// TwinCAT 3 PLC project Fraktal_Press_Demo
// Title: Fraktal_Press_Demo
// Company: fraktal-automation
// Author: fraktal-automation
// ProjectVersion: 0.1.0.10
// Description: CX2030 virtual/physical commissioning example: XTI-linked EK1200/EL1809/EL2809 HAL mapping, two-hand start, interlocked door/part slide, safety aliases, Control On/Off, AUTO/HOME/MANUAL, and model recipes.
// ProgramVersion: 3.1.4026.24
// libraries:
//   Fraktal_Core, 0.25.0.0 (fraktal-automation)
//   Fraktal_Modules, 0.11.0.3 (fraktal-automation)
//   Tc2_MC2, * (Beckhoff Automation GmbH)
//   Tc2_EtherCAT, * (Beckhoff Automation GmbH)
//   Tc2_Standard, * (Beckhoff Automation GmbH)
//   Tc2_System, * (Beckhoff Automation GmbH)
//   Tc3_Module, * (Beckhoff Automation GmbH)
// project tree:
//   00_System/Hardware/ GVL_PressIO.TcGVL, GVL_PressSafety.TcGVL
//   00_System/ GVL_PressCommissioning.TcGVL, MAIN.TcPOU, FB_PressIoDriver.TcPOU, FB_PressControlOnCircuit.TcPOU, FB_PressControlDomain.TcPOU (not stored), FB_PressOutputAuthority.TcPOU (not stored), FB_PressSimulationDriver.TcPOU (not stored)
//   01_PneumaticPress/Sequences/ FB_LD_PressDemoAuto.TcPOU, FB_PressDemoLoadPosition.TcPOU, FB_PressDemoHome.TcPOU, FB_PressDemoChangeover.TcPOU, FB_PressDemoAuto.TcPOU, FB_SFC_PressDemoAuto.TcPOU
//   / PlcTask.TcTTO (not stored)
//   01_PneumaticPress/Release/ FB_PressDemoRelease.TcPOU, FB_LD_PressDemoRelease.TcPOU, FB_PressDemoReleaseState.TcPOU
//   01_PneumaticPress/DUTs/ ST_PressDemoReleaseConditions.TcDUT, ST_PneumaticPressParCfg.TcDUT, ST_PneumaticPressStationCfg.TcDUT, ST_PneumaticPressParCmd.TcDUT (not stored), ST_PneumaticPressOutCmd.TcDUT, ST_PneumaticPressOutImm.TcDUT, E_RenditionLanguage.TcDUT
//   01_PneumaticPress/ PL_PressReasons.TcGVL, FB_PressDemoUnit.TcPOU
//   01_PneumaticPress/Recipes/ FB_PressRecipeCatalog.TcPOU
//   01_PneumaticPress/Io/ FB_PressIoCatalog.TcPOU, GVL_PressFieldbus.TcGVL
// real-time tasks:
//   TASK PlcTask: cycle T#10ms, priority 20, ADS port 350
// I/O:
//   DEVICE =000+S-A610-A1 (EtherCAT) (disabled), AmsNetId 0.0.0.0.2.1
//     =000+S-K010 (EK1200) [EK1200-5000 EtherCAT Power supply (2A E-Bus)]
//       =000+S-K010B1 (EL1809) [EL1809 16Ch. Dig. Input 24V, 3ms]
//       =000+S-K010C1 (EL2809) [EL2809 16Ch. Dig. Output 24V, 0.5A]
//       =000+S-K010D1 (EL6001) [EL6001 Interface (RS232)]
//       =000+S-K010E (EL9011) [EL9011 End Terminal]
// variable links:
//   Fraktal_Press_Demo/Fraktal_Press_Demo Instance <-> =000+S-A610-A1 (EtherCAT)/=000+S-K010 (EK1200)/=000+S-K010B1 (EL1809)
//     PlcTask Inputs/GVL_PressIO._000BS901 <-> Channel 9/_000BS901
//     PlcTask Inputs/GVL_PressIO._000BS902 <-> Channel 13/_000BS902
//     PlcTask Inputs/GVL_PressIO._000K910A <-> Channel 15/_000K910A
//     PlcTask Inputs/GVL_PressIO._000K911_Y32 <-> Channel 14/_000K911_Y32
//     PlcTask Inputs/GVL_PressIO._000MB085A_2 <-> Channel 10/_000MB085A_2
//     PlcTask Inputs/GVL_PressIO._000MB085A_4 <-> Channel 11/_000MB085A_4
//     PlcTask Inputs/GVL_PressIO._101B201A <-> Channel 3/_101B201A
//     PlcTask Inputs/GVL_PressIO._101B202A <-> Channel 5/_101B202A
//     PlcTask Inputs/GVL_PressIO._101B301A <-> Channel 1/_101B301A
//     PlcTask Inputs/GVL_PressIO._101B201B <-> Channel 4/_101B201B
//     PlcTask Inputs/GVL_PressIO._101B202B <-> Channel 6/_101B202B
//     PlcTask Inputs/GVL_PressIO._101B301B <-> Channel 2/_101B301B
//     PlcTask Inputs/GVL_PressIO._101B601 <-> Channel 12/_101B601
//     PlcTask Inputs/GVL_PressIO._101S101 <-> Channel 7/_101S101
//     PlcTask Inputs/GVL_PressIO._101S102 <-> Channel 8/_101S102
//   Fraktal_Press_Demo/Fraktal_Press_Demo Instance <-> =000+S-A610-A1 (EtherCAT)/=000+S-K010 (EK1200)/=000+S-K010C1 (EL2809)
//     PlcTask Outputs/GVL_PressIO._000K911_A1 <-> Channel 11/_000K911_A1
//     PlcTask Outputs/GVL_PressIO._000K951_A1 <-> Channel 10/_000K951_A1
//     PlcTask Outputs/GVL_PressIO._101K201A <-> Channel 3/_101K201A
//     PlcTask Outputs/GVL_PressIO._101K202A <-> Channel 5/_101K202A
//     PlcTask Outputs/GVL_PressIO._101K301A <-> Channel 1/_101K301A
//     PlcTask Outputs/GVL_PressIO._101K201B <-> Channel 4/_101K201B
//     PlcTask Outputs/GVL_PressIO._101K202B <-> Channel 6/_101K202B
//     PlcTask Outputs/GVL_PressIO._101K301B <-> Channel 2/_101K301B
//     PlcTask Outputs/GVL_PressIO._101P101 <-> Channel 7/_101P101
//     PlcTask Outputs/GVL_PressIO._101P102 <-> Channel 8/_101P102

// ---- 01_PneumaticPress/DUTs/ST_PressDemoReleaseConditions.TcDUT
// Core §7.2/§3.12 - the press's named release conditions, as PUBLISHED.
// Filled every scan from whichever rendition RELEASE_LANGUAGE selects, so a
// browsing client always reads the conditions that are actually being
// evaluated. Before this, the ST component was the published one and was
// never evaluated while LADDER_DIAGRAM was selected: every flag sat at its
// initial FALSE whatever the machine was doing - state nobody computes,
// published as if it were a claim.
TYPE ST_PressDemoReleaseConditions :
STRUCT
    ModeStartAirPressureOk : BOOL;
    RamGuardClosed    : BOOL;
    RamSlideInside    : BOOL;
    RamDevicesHealthy : BOOL;
    RamAirPressureOk  : BOOL;
    RamTwoHandHeld    : BOOL;
    RamControlPowerOn : BOOL;
END_STRUCT
END_TYPE

// ---- 01_PneumaticPress/DUTs/ST_PneumaticPressParCfg.TcDUT
// Core §3.8 ParCfg (SchemaVersion first; adding a member = schema change).
// v2 adds the §8.11 performance references: per-model ideal cycle (OEE
// Performance denominator, §8.5.1) and the WORK-time degradation baseline
// (§8.11.4(d); 0 = watch off).
//
// v3 REMOVES RequireTwoHandStart. It was recipe data in name only - every one of
// the four catalog records set it TRUE - and §3.8a's test is whether the value
// changes with the model. It does not: it answers whether this CELL's risk
// assessment demands a two-hand start, which is deployment data and now lives in
// ST_PneumaticPressStationCfg. A recipe that could switch it off would let a
// changeover quietly remove a required operator protection.
//
// TransferSettleTime deliberately STAYED. Its catalog values genuinely differ per
// model (80/100/120/150 ms): a heavier steel blank settles on the slide more
// slowly than a plastic one, so it is a fact about the part, not the mechanism.
TYPE ST_PneumaticPressParCfg :
STRUCT
    SchemaVersion       : UINT := 3;
    PressSettleTime     : TIME := T#500MS;
    TransferSettleTime  : TIME := T#100MS;
    IdealCycleMs        : UDINT := 0;    // §8.5.1 — 0 = Performance not computed
    BaselineWorkMs      : UDINT := 0;    // §8.11.4(d) — 0 = degradation watch off
END_STRUCT
END_TYPE

// ---- 01_PneumaticPress/DUTs/ST_PneumaticPressStationCfg.TcDUT
// Core §3.8a/§3.8b — what this PRESS is, as opposed to what the current product
// needs. Both members were assessed against one question: does the value change
// when the MODEL changes?
//
//   RequireTwoHandStart came OUT of ST_PneumaticPressParCfg. It was recipe data
//   in name only - all four catalog records set it TRUE - and it answers a
//   question about the CELL: does this installation's risk assessment demand a
//   two-hand start? A model recipe able to switch it off would let a changeover
//   quietly remove a required operator protection, which is not a decision a
//   product record should be able to take. (The certified two-hand evaluation
//   stays in TwinSAFE regardless, §9.8; this flag selects whether the AUTO cycle
//   WAITS for it, and can never weaken the safety function itself.)
//
//   StallGuardMs is the step guard for a step that declares no ExpectedTime
//   (§6.9). How long a pneumatic motion may take before it counts as stalled is
//   a fact about this machine's cylinders and air supply, not about the part.
//
// SchemaVersion is FIRST and mandatory (§3.8b). Version 0 means never written, so
// a first boot initializes silently; any other unrecognized version means a real
// image was rejected, and FB_ModuleBase.M_RestoreStationCfg reports it for the
// root to annunciate with this Unit's canonical path.
TYPE ST_PneumaticPressStationCfg :
STRUCT
    SchemaVersion       : UINT;    // 0 = never written; 1 = this layout
    RequireTwoHandStart : BOOL;    // cell risk-assessment policy, not recipe data
    StallGuardMs        : UDINT;   // §6.9 step guard when a step declares none
END_STRUCT
END_TYPE

// ---- 01_PneumaticPress/DUTs/ST_PneumaticPressOutCmd.TcDUT
TYPE ST_PneumaticPressOutCmd :
STRUCT
    // §3.12 — OutCmd is what a COMMAND PRODUCED, latched until the next command.
    // Both of these are genuine command results: a cycle ran, a changeover ran.
    // `Homed` used to live here and does not any more - being at the home position
    // is not something a command produced, it is something that is either true now
    // or not, so it is derived state (OutImm.Homed) recomputed every scan.
    CycleCompleted : BOOL;
    ChangeoverCompleted : BOOL;
END_STRUCT
END_TYPE

// ---- 01_PneumaticPress/DUTs/ST_PneumaticPressOutImm.TcDUT
TYPE ST_PneumaticPressOutImm :
STRUCT
    // Only facts the Unit DERIVES. A child's own state is read on the child
    // (PressRam.OutImm.Retracted, ...), never copied here under a second name (O9).
    //
    // §3.12 derived state: TRUE while the machine IS at its reference position.
    // As a latched command result it went on claiming "homed" after an operator
    // jogged an axis off home in MANUAL, because no sequence ran to clear it.
    Homed           : BOOL;
    // TRUE while a two-hand press would start a cycle: buttons armed, the control
    // domain ready, a part loaded and air present. Drives the pushbutton lamps.
    TwoHandStartReady : BOOL;
END_STRUCT
END_TYPE

// ---- 01_PneumaticPress/DUTs/E_RenditionLanguage.TcDUT
// Which language a parallel rendition of the same engineering is written in.
// The internal press bench carries the AUTO chain three times and the release
// engineering twice — the same behaviour in a second language is a
// demonstration of §5.5/§6.8 language parity, not §1.1 O9 duplication.
// FB_PressDemoUnit selects one of each; the compiler folds the branches the
// selection does not take, so the unselected renditions are inert.
//
// ONE type for both selections on purpose: a value has to mean the same
// language wherever it appears. The release engineering has no
// SEQUENTIAL_FUNCTION_CHART rendition — SFC is a sequence language and has
// nothing to say about a permissive — so that member is simply never selected
// there. The gap is deliberate; it is not an invitation to reuse the value for
// something else.
//
// The members are spelled out rather than abbreviated because 'ST' is a
// reserved word (the IL store operator). As an enumeration member it desyncs
// the parser and cascades misleading errors onto innocent lines (lint C2).
{attribute 'qualified_only'}
TYPE E_RenditionLanguage :
(
    STRUCTURED_TEXT           := 0,   // §6.8 reference form: CASE _step OF + M_Advance
    SEQUENTIAL_FUNCTION_CHART := 1,   // native XAE chart; sequences only
    LADDER_DIAGRAM            := 2    // rung-per-state integer machine over _step
) DINT;
END_TYPE

// ---- 00_System/Hardware/GVL_PressIO.TcGVL
{attribute 'qualified_only'}
// CX2030 local EtherCAT process image, reconciled with the supplied XTI export.
// TcLinkTo owns the physical link by exact terminal/channel/PDO-entry name;
// AT %I*/%Q* keeps the compiler-selected process-image offset non-positional.
VAR_GLOBAL
    // =000+S-K010B1 (EL1809) inputs
    {attribute 'TcLinkTo' := 'TIIB[=000+S-K010B1 (EL1809)]^Channel 1^_101B301A'}
    _101B301A AT %I* : BOOL;       // Ch1 feeder retracted = logical slide INSIDE
    {attribute 'TcLinkTo' := 'TIIB[=000+S-K010B1 (EL1809)]^Channel 2^_101B301B'}
    _101B301B AT %I* : BOOL;       // Ch2 feeder extended  = logical slide OUTSIDE
    {attribute 'TcLinkTo' := 'TIIB[=000+S-K010B1 (EL1809)]^Channel 3^_101B201A'}
    _101B201A AT %I* : BOOL;       // Ch3 door closed
    {attribute 'TcLinkTo' := 'TIIB[=000+S-K010B1 (EL1809)]^Channel 4^_101B201B'}
    _101B201B AT %I* : BOOL;       // Ch4 door open
    {attribute 'TcLinkTo' := 'TIIB[=000+S-K010B1 (EL1809)]^Channel 5^_101B202A'}
    _101B202A AT %I* : BOOL;       // Ch5 press down
    {attribute 'TcLinkTo' := 'TIIB[=000+S-K010B1 (EL1809)]^Channel 6^_101B202B'}
    _101B202B AT %I* : BOOL;       // Ch6 press up
    {attribute 'TcLinkTo' := 'TIIB[=000+S-K010B1 (EL1809)]^Channel 7^_101S101'}
    _101S101  AT %I* : BOOL;       // Ch7 right two-hand raw button
    {attribute 'TcLinkTo' := 'TIIB[=000+S-K010B1 (EL1809)]^Channel 8^_101S102'}
    _101S102  AT %I* : BOOL;       // Ch8 left two-hand raw button
    {attribute 'TcLinkTo' := 'TIIB[=000+S-K010B1 (EL1809)]^Channel 10^_000MB085A_2'}
    _000MB085A_2 AT %I* : BOOL;    // Ch10 compressed air below 0.3 bar
    {attribute 'TcLinkTo' := 'TIIB[=000+S-K010B1 (EL1809)]^Channel 11^_000MB085A_4'}
    _000MB085A_4 AT %I* : BOOL;    // Ch11 compressed air above 4.5 bar
    {attribute 'TcLinkTo' := 'TIIB[=000+S-K010B1 (EL1809)]^Channel 12^_101B601'}
    _101B601 AT %I* : BOOL;        // Ch12 part present
    // N54 D2 operator buttons. Free EL1809 channels were 9/13/16; 9 and 13 are
    // assigned here. The TcLinkTo names MUST match the terminal channel names in
    // XAE - confirm the physical wiring before trusting these.
    {attribute 'TcLinkTo' := 'TIIB[=000+S-K010B1 (EL1809)]^Channel 9^_000BS901'}
    _000BS901 AT %I* : BOOL;       // Ch9  IsControlOnButtonPressed  (=000+B-S901:14)
    {attribute 'TcLinkTo' := 'TIIB[=000+S-K010B1 (EL1809)]^Channel 13^_000BS902'}
    _000BS902 AT %I* : BOOL;       // Ch13 IsControlOffButtonPressed (=000+B-S902:14)
    {attribute 'TcLinkTo' := 'TIIB[=000+S-K010B1 (EL1809)]^Channel 14^_000K911_Y32'}
    _000K911_Y32 AT %I* : BOOL;    // Ch14 Control On feedback
    {attribute 'TcLinkTo' := 'TIIB[=000+S-K010B1 (EL1809)]^Channel 15^_000K910A'}
    _000K910A AT %I* : BOOL;       // Ch15 E-stop PRESSED (=000+S1-K910A:14); NORMALLY OPEN on this
                                   // demo rig: TRUE = actuated. NOT fail-safe - production needs NC.

    // =000+S-K010C1 (EL2809) outputs
    {attribute 'TcLinkTo' := 'TIIB[=000+S-K010C1 (EL2809)]^Channel 1^_101K301A'}
    _101K301A AT %Q* : BOOL;       // Ch1 feeder backward = move inside
    {attribute 'TcLinkTo' := 'TIIB[=000+S-K010C1 (EL2809)]^Channel 2^_101K301B'}
    _101K301B AT %Q* : BOOL;       // Ch2 feeder forward  = move outside
    {attribute 'TcLinkTo' := 'TIIB[=000+S-K010C1 (EL2809)]^Channel 3^_101K201A'}
    _101K201A AT %Q* : BOOL;       // Ch3 close door
    {attribute 'TcLinkTo' := 'TIIB[=000+S-K010C1 (EL2809)]^Channel 4^_101K201B'}
    _101K201B AT %Q* : BOOL;       // Ch4 open door
    {attribute 'TcLinkTo' := 'TIIB[=000+S-K010C1 (EL2809)]^Channel 5^_101K202A'}
    _101K202A AT %Q* : BOOL;       // Ch5 press downward
    {attribute 'TcLinkTo' := 'TIIB[=000+S-K010C1 (EL2809)]^Channel 6^_101K202B'}
    _101K202B AT %Q* : BOOL;       // Ch6 press upward
    {attribute 'TcLinkTo' := 'TIIB[=000+S-K010C1 (EL2809)]^Channel 7^_101P101'}
    _101P101  AT %Q* : BOOL;       // Ch7 right two-hand lamp
    {attribute 'TcLinkTo' := 'TIIB[=000+S-K010C1 (EL2809)]^Channel 8^_101P102'}
    _101P102  AT %Q* : BOOL;       // Ch8 left two-hand lamp
    {attribute 'TcLinkTo' := 'TIIB[=000+S-K010C1 (EL2809)]^Channel 10^_000K951_A1'}
    _000K951_A1 AT %Q* : BOOL;     // Ch10 SwitchControlOn functional request
    {attribute 'TcLinkTo' := 'TIIB[=000+S-K010C1 (EL2809)]^Channel 11^_000K911_A1'}
    _000K911_A1 AT %Q* : BOOL;     // Ch11 EnableControlOn functional request

    // =000+S-K010D1 (EL6001) RS232 serial interface.
    //
    // The terminal is on the bus and was previously unmapped, so it appeared in the
    // topology as a node with no channels: an operator diagnosing a dead serial link
    // had nothing to look at. Nothing in this demo speaks a serial protocol yet - the
    // process image is mapped so the card is visible, forceable and diagnosable like
    // every other node, which is what the §10.5.1 bus view is for.
    //
    // [!] NOT LINKED YET. The guessed default 3-byte PDO names (0x1A00/0x1600) were
    // wrong - XAE reports `TIIB[=000+S-K010D1 (EL6001)]^Inputs^Status` not found, so
    // this terminal is on a different PDO assignment. The variables and their §10.5.1
    // topology channels stay (the card is published and visible); only the process
    // image link is missing. To finish: open the terminal's Process Data tab, read the
    // actual PDO entry names, and restore a TcLinkTo per variable. A wrong TcLinkTo
    // fails the build loudly, which is the right failure mode - it is why these are
    // absent rather than guessed a second time.
    _000K010D1_Status AT %I* : USINT;    // serial status byte
    _000K010D1_DataIn0 AT %I* : USINT;
    _000K010D1_DataIn1 AT %I* : USINT;
    _000K010D1_DataIn2 AT %I* : USINT;
    _000K010D1_Ctrl AT %Q* : USINT;      // serial control byte
    _000K010D1_DataOut0 AT %Q* : USINT;
    _000K010D1_DataOut1 AT %Q* : USINT;
    _000K010D1_DataOut2 AT %Q* : USINT;
END_VAR

// ---- 00_System/Hardware/GVL_PressSafety.TcGVL
{attribute 'qualified_only'}
// Read-only aliases to results produced outside the standard PLC by TwinSAFE
// or a validated external safety system. They intentionally default FALSE so
// physical mode cannot energize until commissioning supplies every result.
// These variables do not themselves implement a safety function.
VAR_GLOBAL
    _EStopOk               AT %I* : BOOL;
    _GuardClosed           AT %I* : BOOL;
    _TwoHandActive         AT %I* : BOOL;
    _PneumaticPermit       AT %I* : BOOL;
    _SafetyFieldbusHealthy AT %I* : BOOL;
    _StandardIoHealthy     AT %I* : BOOL;
END_VAR

// ---- 00_System/GVL_PressCommissioning.TcGVL
{attribute 'qualified_only'}
// Deployment-owned access-provider bootstrap. Secrets deliberately have no
// source default and are excluded from OPC UA. Write a PIN here in the target's
// controlled commissioning workflow: MAIN registers it as a salted hash in the same
// scan and clears it, so no PIN is retained as text (§14). Provision users before
// locking the PLC policy.
VAR_GLOBAL PERSISTENT
    {attribute 'OPC.UA.DA' := '0'}
    OperatorPin   : STRING(32);
    {attribute 'OPC.UA.DA' := '0'}
    TechnicianPin : STRING(32);
    {attribute 'OPC.UA.DA' := '0'}
    AdminPin      : STRING(32);
END_VAR

// ---- 01_PneumaticPress/PL_PressReasons.TcGVL
{attribute 'qualified_only'}
// Core §8.8 band constants for THIS project: pneumatic press 12000-12999.
// Project codes deliberately sit outside the shipped registry, so a message
// raised with one keeps the severity and category the step chose.
VAR_GLOBAL CONSTANT
    PRESS_TWO_HAND_RELEASED : DINT := 12001;   // released mid-motion: cycle aborted, no damage
END_VAR

// ---- 01_PneumaticPress/Io/GVL_PressFieldbus.TcGVL
{attribute 'qualified_only'}
// Owner-local, bounded publication of the demo's physical CX2030 I/O tree.
// ST_IoChannel.Name is always the exact electrical-list/schematic tag.
VAR_GLOBAL
    {attribute 'OPC.UA.DA' := '1'}
    Topology : ST_FieldbusTopology;
END_VAR

// ---- 00_System/MAIN.TcPOU
// Virtual-commissioning application for one pneumatic press Unit.
// IMPORTANT: the Safe* values below simulate TwinSAFE outputs only. A deployed
// machine maps certified E-stop/two-hand/guard/safe-valve results from TwinSAFE.
PROGRAM MAIN
VAR
    RecipeCatalog : FB_PressRecipeCatalog;
    // §3.8b - WHERE this station's retained data lives is a project decision, made
    // here once: the press keeps its station, line and model data, its saved
    // parameter sets and its local users as files in DATA_FOLDER. A station with
    // no usable file system declares FB_RetainPersistMedium instead and nothing
    // else changes (users then stay in the Boot directory: a credential never goes
    // to a symbol-readable medium). On an IPC image with a write filter the folder
    // must be excluded, or every write reverts at the next boot.
    Storage : FB_FilePersistMedium;
    // §3.8b - named parameter sets on the same medium: one readable JSON-lines
    // file per saved set.
    ConfigStore : FB_MediumConfigStore;
    PartCarrier : FB_LocalPartCarrier;    // §3.16.2 BY_POSITION identity + local result ring
    AccessUsers : FB_LocalAccessProvider; // §7.7 commissioning user/PIN table
    // TF6100 TMC-Filtered publication starts at the deployed root instance.
    // The marker is inherited by PneumaticPress's published child symbols.
    {attribute 'OPC.UA.DA' := '1'}
    PneumaticPress : FB_PressDemoUnit;
    // §3.8e - the line this press stands on, and the OWNER of its data (the shift
    // calendar, §8.5.2). A line is no Unit and no module of one: it sits here,
    // beside the roots, like the control domain, and each root on the line
    // references it (SetLine) and presents its values as that root's line data.
    // A second station on this line would host a MIRROR fed through I_LineSource.
    PressLine : FB_LineDataV3;
    IoCatalog : FB_PressIoCatalog;
    IoDriver : FB_PressIoDriver;
    // Core §7.5.1 — this station's commissioning/engineering gate register.
    // Every gate below is a VAR CONSTANT of this program, so the register is
    // decided at build time and cannot be edited on a running machine. While it
    // holds anything, every root Unit carries the standing §7.5.2 annunciation.
    EngineeringMode : FB_EngineeringMode;
    ControlDomain : FB_PressControlDomain;
    OutputAuthority : FB_PressOutputAuthority;
    SimulationDriver : FB_PressSimulationDriver;
    PressHal, DoorHal, SlideHal : ST_CylinderHal;
    TwoHandHal : ST_TwoHandHal;
    PowerHal : ST_PowerGroupHal;
    PartPresentHal : ST_DigitalInputHal;
    AirPressureHal : ST_AirPressureHal;
    HealthProbe : FB_TcSystemHealthProbe;
    HealthConfig : ST_SystemHealthParCfg;
    HealthCpuLoadPct : LREAL;
    HealthMemoryAvailableMb : UDINT;
    HealthTimeSource : STRING(32);
    TaskIndex : Tc2_System.GETCURTASKINDEX;
    TaskCycleUs : UDINT;
    InitialModel : ST_ModelId;
    Plate : ST_Nameplate;
    Init : BOOL;
    // Read-only MIRRORS of the commissioning gates (see the VAR CONSTANT block).
    // They exist only so the gate state stays visible over ADS/OPC UA: the
    // compiler inlines constants, which may publish no symbol at all, and losing
    // that visibility would remove the fastest way to diagnose "no output moves".
    // They are reassigned from the constants every cycle and nothing reads them,
    // so writing one online is inert - the constant remains the only authority.
    UseSimulation : BOOL;
    ControlCircuitMappingConfirmed : BOOL;
    // §10.5.1 demand gate, written by the HMI while its fieldbus page is open.
    // FALSE parks the EtherCAT master scan (no ADS traffic for a view nobody is
    // watching); the last read states are held, never falsified.
    FieldbusViewActive : BOOL;

    // Simulation controls. E-stop is normally closed: TRUE = healthy circuit.
    SimEStopNc : BOOL := TRUE;
    SimControlOnButton : BOOL;
    SimControlOffButton : BOOL;
    SimLeftButton : BOOL;
    SimRightButton : BOOL;
    SimSafetyValveOk : BOOL := TRUE;
    SimFieldbusHealthy : BOOL := TRUE;
    SimPartPresent : BOOL := TRUE;
    SimAirPressureOk : BOOL := TRUE;
    SafeEStopOk : BOOL;
    SafeGuardClosed : BOOL;
    SafeTwoHandActive : BOOL;
    SafePneumaticPermit : BOOL;
    SafetyFieldbusHealthy : BOOL;
    StandardIoHealthy : BOOL;
    RawEStopHealthy : BOOL;
    LampsOn : BOOL;
    ControlOnEdge : R_TRIG;
    ControlOffEdge : R_TRIG;
    ControlOnAdopted : R_TRIG;   // rising edge of the relay chain's feedback
END_VAR
VAR CONSTANT
    // COMMISSIONING GATES - deliberately CONSTANT so they cannot be flipped
    // online. Defeating a gate must be a source change plus a download: a
    // reviewable, auditable act, not a live write from an HMI or ADS client.
    //
    // TRUE makes MAIN call M_ClearOutputs() every cycle, so no physical output
    // is ever energized while the simulation driver animates the plant.
    USE_SIMULATION : BOOL := FALSE;
    // FALSE makes M_WriteOutputs force _000K951_A1 and _000K911_A1 FALSE every
    // cycle. Control On then cannot energize, the hardwired N54 D2 relay chain
    // never closes, and NOTHING moves - even though the cylinder coils are
    // written unconditionally. Set TRUE only after verifying the K951/K911
    // electrical semantics on the cabinet; per N54 D2 SwitchControlOn and
    // EnableControlOn are distinct signals.
    CONTROL_CIRCUIT_MAPPING_CONFIRMED : BOOL := TRUE;
    // §G.4a - does THIS bench have a safety-rated enabling device for manual
    // motion? It does not: the Xvi is an 80 N magnetic linear motor standing on
    // the desk, outside the press. Declaring that here makes the axis's
    // StationCfg say the same thing, and the §7.5 gate below makes the machine
    // announce the departure for as long as it is true. A real cell with a
    // person inside it sets this TRUE and the §G.4a rule applies unchanged.
    JOG_ENABLE_DEVICE_REQUIRED : BOOL := FALSE;
END_VAR
VAR CONSTANT
    // §3.8b - this station's data folder (FB_FilePersistMedium, PATH_GENERIC).
    DATA_FOLDER : STRING(160) := 'C:\ProgramData\Fraktal\PressDemo\';
END_VAR

// Mirror the compile-time gates so they remain observable (see declaration).
UseSimulation := USE_SIMULATION;
ControlCircuitMappingConfirmed := CONTROL_CIRCUIT_MAPPING_CONFIRMED;

IF NOT Init THEN
    Init := TRUE;
    // Initial mechanically safe/load position: ram up, door open, slide outside.
    PressHal.RetractedFb := TRUE;
    DoorHal.RetractedFb := TRUE;
    SlideHal.RetractedFb := TRUE;
    RecipeCatalog.Setup(UnitRef := PneumaticPress);
    PneumaticPress.Setup(Name := 'PneumaticPress', PressHal := PressHal, DoorHal := DoorHal,
        SlideHal := SlideHal, TwoHandHal := TwoHandHal, PowerHal := PowerHal,
        PartPresentHal := PartPresentHal, AirPressureHal := AirPressureHal,
        Recipe := RecipeCatalog.Provider);
    PressLine.Setup(Name := 'PressLine', LineId := 'PRESS-LINE-1',
        Role := E_LineRole.OWNER, Source := 0, StaleAfterMs := 0);
    PneumaticPress.SetLine(pLine := ADR(PressLine));
    // §7.5.1 — declare this project's own gates. Passing the CONSTANT as `Active`
    // is the point: an inactive gate registers nothing, so a production build
    // publishes an empty register, annunciates nothing, and exposes no gated
    // surface at all. Passing a runtime variable here would defeat §7.5.1.
    EngineeringMode.M_Declare(Name := 'USE_SIMULATION',
        DescriptionKey := 'std.engineering.simulation', Active := USE_SIMULATION);
    EngineeringMode.M_Declare(Name := 'CONTROL_CIRCUIT_UNCONFIRMED',
        DescriptionKey := 'std.engineering.controlCircuitUnconfirmed',
        Active := NOT CONTROL_CIRCUIT_MAPPING_CONFIRMED);
    EngineeringMode.M_Declare(Name := 'JOG_ENABLE_DEVICE_NOT_REQUIRED',
        DescriptionKey := 'std.engineering.jogEnableDeviceNotRequired',
        Active := NOT JOG_ENABLE_DEVICE_REQUIRED);
    // Wiring the register also declares the framework's own OUTPUT_FORCING gate
    // from PL_FraktalEngineering, so forcing can never be armed without being
    // annunciated. It must precede IoCatalog.Setup, which reads ForcingActive to
    // decide whether any channel is published as Forceable at all.
    PneumaticPress.SetEngineeringMode(Mode := EngineeringMode);
    IoDriver.Setup(UnitRef := PneumaticPress);
    IoCatalog.Setup(UnitRef := PneumaticPress, Engineering := EngineeringMode);
    // §10.5.1 — the catalog owns the approved channel join, so it is what
    // resolves a force request; the Unit only routes an already-authorized one.
    PneumaticPress.SetIoCatalog(Catalog := IoCatalog);
    ControlDomain.Setup(UnitRef := PneumaticPress);
    SimulationDriver.Setup(PressHal := PressHal, DoorHal := DoorHal, SlideHal := SlideHal);
    InitialModel.ModelCode := 'ALUMINUM';
    PneumaticPress.SetModel(Id := InitialModel);
    Plate.ProductUri := 'urn:fraktal:demo:pneumatic-press:2026-0001';
    Plate.ManufacturerName := 'Fraktal Example Project';
    Plate.ProductDesignation := 'Pneumatic Press Training Cell';
    Plate.SerialNumber := 'PRESS-DEMO-2026-0001';
    Plate.YearOfConstruction := '2026';
    Plate.SoftwareVersion := 'Fraktal Press Demo 0.1';
    PneumaticPress.SetNameplate(Plate := Plate);
    // §8.9 standard reason metadata is generated and manifest-served by the Unit.
    // §3.16 traceability: station-local BY_POSITION serials; RFID/host substitutes later
    PartCarrier.Setup(UidPrefix := 'PRESS-2026-');
    PneumaticPress.SetPartCarrier(Carrier := PartCarrier);
    // §3.8b — the medium, then everything kept on it. Composition-root wiring, no
    // per-value glue: every capability any module in this tree registered is in
    // the station, line and model documents and in every saved set already.
    Storage.Setup(Folder := DATA_FOLDER, Where := Tc2_System.PATH_GENERIC);
    ConfigStore.Setup(Medium := Storage, KeyPrefix := 'PneumaticPress.sets');
    PneumaticPress.SetConfigStore(Store := ConfigStore);
    PneumaticPress.SetPersistMedium(Medium := Storage);
    // §3.8b — this press declares the STRICT restore policy. Its station data
    // today is the two-hand requirement and the step stall guard, and the
    // two-hand requirement is the reason: losing it would mean a machine that
    // presents itself as commissioned while no longer waiting for the start
    // control this cell's risk assessment requires. DEFAULTS_AND_ANNUNCIATE is
    // the shipped default and is right for a station whose lost values are
    // conveniences; this one's are not.
    //
    // The PartFeed axis's taught position is NOT in this set. FB_AxisCM
    // registers it (Annex G §G.4b), but PartFeed is neither bound by
    // ConfigurePartFeedAxis nor registered as a child of this Unit while no NC
    // axis exists in the System Manager — so it is outside the walk, and a
    // station set taken here does not contain it. It joins the set the day the
    // axis is linked, with no change to this line.
    PneumaticPress.SetConfigRestorePolicy(
        Policy := E_ConfigRestorePolicy.BLOCK_UNTIL_ACKNOWLEDGED);
    // §G.4a - the axis's own retained StationCfg is the authority; this states
    // the bench's fact into it. Stamps the schema version too, so the value
    // survives the axis's later Setup/restore rather than being defaulted over.
    IF NOT JOG_ENABLE_DEVICE_REQUIRED THEN
        PneumaticPress.PartFeed.SetJogRequiresEnable(Required := FALSE);
    END_IF
    // §7.7(c) - the user table (names and salted PIN hashes) on the same medium.
    AccessUsers.M_UseMedium(Medium := Storage);
    AccessUsers.M_UseKey(Key := 'PneumaticPress.users');
    PneumaticPress.Access.Setup(Provider := AccessUsers, pAlarmLog := ADR(PneumaticPress.AlarmLog));
    TaskIndex();
    TaskCycleUs := _TaskInfo[TaskIndex.index].CycleTime / 10;
    HealthConfig.MaxTaskCycleUs := TaskCycleUs + 2000;
    HealthProbe.M_UseWindowsTime(Enabled := NOT USE_SIMULATION,
        FilePath := PL_Fraktal.WINDOWS_CLOCK_SAMPLE_FILE, MaximumSampleAge := T#90S,
        MaximumSyncAgeSeconds := 7200, MaximumOffsetUs := HealthConfig.MaxTimeOffsetUs);
    // §8.12/§10.5 - the real profile measures controller/IPC health through the
    // Beckhoff Device Manager and the bus through the EtherCAT master's own state,
    // frame and CRC counters; simulation keeps the synthetic explicit inputs.
    HealthProbe.M_UseIpcDiagnostics(Enabled := NOT USE_SIMULATION);
    IF NOT USE_SIMULATION THEN
        HealthProbe.M_UseEtherCatMaster(pBus := IoDriver.M_BusHealth());
    END_IF
    HealthConfig.MaxTaskJitterUs := 2000;
    HealthConfig.RequireFieldbus := TRUE;
    HealthConfig.RequireDcSync := FALSE;
    HealthConfig.RequireTimeSync := TRUE;
END_IF

// §7.7/§14: a PIN is deployment configuration, never a source literal. Write one
// into GVL_PressCommissioning (XAE watch window) and it is registered as a salted
// hash in this scan and wiped: no PIN is retained as text, and the persistent user
// table keeps the user across restarts. Provision users before raising a threshold.
IF GVL_PressCommissioning.OperatorPin <> '' THEN
    AccessUsers.Register(User := 'operator', Pin := GVL_PressCommissioning.OperatorPin,
        Level := E_AccessLevel.OPERATOR);
    GVL_PressCommissioning.OperatorPin := '';
END_IF
IF GVL_PressCommissioning.TechnicianPin <> '' THEN
    AccessUsers.Register(User := 'tech', Pin := GVL_PressCommissioning.TechnicianPin,
        Level := E_AccessLevel.TECHNICIAN);
    GVL_PressCommissioning.TechnicianPin := '';
END_IF
IF GVL_PressCommissioning.AdminPin <> '' THEN
    AccessUsers.Register(User := 'admin', Pin := GVL_PressCommissioning.AdminPin,
        Level := E_AccessLevel.ADMIN);
    GVL_PressCommissioning.AdminPin := '';
END_IF

// Ordinary simulated local station buttons. The worksheet does not list real
// Control On/Off input buttons; physical operation therefore uses HMI requests
// until those devices are identified. Control Off wins simultaneous edges.
// Source the Control On/Off edges from the REAL buttons on a live machine, and
// from the simulated ones only under USE_SIMULATION. Previously both edges were
// ANDed with USE_SIMULATION, so on hardware neither could ever fire and the
// machine had no headless Control On path at all.
IF USE_SIMULATION THEN
    ControlOnEdge(CLK := SimControlOnButton);
    ControlOffEdge(CLK := SimControlOffButton);
ELSE
    ControlOnEdge(CLK := IoDriver.ControlOnButton);
    ControlOffEdge(CLK := IoDriver.ControlOffButton);
END_IF
IF ControlOffEdge.Q THEN
    PneumaticPress.RequestLocalControl(ControlOn := FALSE);
ELSIF ControlOnEdge.Q THEN
    PneumaticPress.RequestLocalControl(ControlOn := TRUE);
END_IF
// Adopt the relay chain's established state: it is the authority. Without this
// the PLC can sit with no power request while K911_Y32 shows control is already
// ON (observed on the press), leaving PLC and hardware permanently out of step.
// One-shot: re-issuing POWER_ON every scan would re-fault the power group on
// any momentary permit dip and spam the event log. Latch on the feedback's
// rising edge only, and re-arm the latch when control drops away.
ControlOnAdopted(CLK := PowerHal.PowerFeedback);
IF NOT USE_SIMULATION AND ControlOnAdopted.Q AND NOT ControlOffEdge.Q THEN
    PneumaticPress.RequestLocalControl(ControlOn := TRUE);
END_IF

IF USE_SIMULATION THEN
    SimulationDriver.M_ReadInputs(DoorHal := DoorHal, TwoHandHal := TwoHandHal,
        PowerHal := PowerHal, PartPresentHal := PartPresentHal,
        AirPressureHal := AirPressureHal, RawEStopHealthy := RawEStopHealthy,
        SafeEStopOk := SafeEStopOk, SafeGuardClosed := SafeGuardClosed,
        SafeTwoHandActive := SafeTwoHandActive,
        SafePneumaticPermit := SafePneumaticPermit,
        SafetyFieldbusHealthy := SafetyFieldbusHealthy,
        StandardIoHealthy := StandardIoHealthy, SimEStopNc := SimEStopNc,
        SimLeftButton := SimLeftButton, SimRightButton := SimRightButton,
        SimSafetyValveOk := SimSafetyValveOk,
        SimFieldbusHealthy := SimFieldbusHealthy,
        SimPartPresent := SimPartPresent, SimAirPressureOk := SimAirPressureOk,
        PowerRequested := PowerHal.EnableRequestOut);
ELSE
    // The project Hardware Driver is the only raw process-image consumer.
    IoDriver.M_ReadInputs(PressHal := PressHal, DoorHal := DoorHal,
        SlideHal := SlideHal, TwoHandHal := TwoHandHal, PowerHal := PowerHal,
        PartPresentHal := PartPresentHal, AirPressureHal := AirPressureHal,
        RawEStopHealthy := RawEStopHealthy, SafeEStopOk := SafeEStopOk,
        SafeGuardClosed := SafeGuardClosed, SafeTwoHandActive := SafeTwoHandActive,
        SafePneumaticPermit := SafePneumaticPermit,
        SafetyFieldbusHealthy := SafetyFieldbusHealthy,
        StandardIoHealthy := StandardIoHealthy);
END_IF
TwoHandHal.SafeActive := SafeTwoHandActive;
TwoHandHal.FieldbusHealthy := SafetyFieldbusHealthy;
PowerHal.SafetyPermit := SafePneumaticPermit;
PowerHal.FieldbusHealthy := StandardIoHealthy;

ControlDomain.M_Update(SafeEStopOk := SafeEStopOk,
    SafeGuardClosed := SafeGuardClosed, SafeTwoHandActive := SafeTwoHandActive,
    SafePneumaticPermit := SafePneumaticPermit,
    SafetyFieldbusHealthy := SafetyFieldbusHealthy,
    StandardIoHealthy := StandardIoHealthy, RawEStopHealthy := RawEStopHealthy,
    PowerFeedback := PowerHal.PowerFeedback,
    PowerRequested := PowerHal.EnableRequestOut,
    TwoHandFieldbusHealthy := TwoHandHal.FieldbusHealthy);
PneumaticPress.ControlDomain := ControlDomain.Status;

// §2.7/§8.12: in the real profile the probe measures the target itself - Windows
// Time through the local observer, controller/IPC metrics through the Device
// Manager, the bus through the EtherCAT master - and those groups ignore the
// explicit inputs below, which remain the simulation profile's synthetic values.
IF USE_SIMULATION THEN
    HealthCpuLoadPct := 25.0;
    HealthMemoryAvailableMb := UDINT#1024;
    HealthTimeSource := 'SIMULATED';
ELSE
    HealthCpuLoadPct := 0.0;
    HealthMemoryAvailableMb := UDINT#0;
    HealthTimeSource := 'WINDOWS/W32TIME';
END_IF
TaskIndex();
TaskCycleUs := _TaskInfo[TaskIndex.index].CycleTime / 10;
HealthProbe.Cyclic(ExpectedCycleUs := TaskCycleUs,
    ExternalTaskOverrun := _TaskInfo[TaskIndex.index].CycleTimeExceeded,
    ControllerAvailable := USE_SIMULATION,
    CpuLoadPct := HealthCpuLoadPct,
    MemoryAvailableMb := HealthMemoryAvailableMb,
    IpcAvailable := FALSE, IpcTemperatureC := 0.0,
    FanHealthy := TRUE, StorageHealthPct := 100.0,
    FieldbusAvailable := TRUE, FieldbusMasterHealthy := StandardIoHealthy,
    LostFrameCount := 0, SlaveErrorCount := 0,
    DcAvailable := USE_SIMULATION, DcSynchronized := USE_SIMULATION,
    TimeAvailable := USE_SIMULATION, TimeSynchronized := USE_SIMULATION,
    TimeSource := HealthTimeSource,
    TimeOffsetUs := 0, LastSyncAt := F_Now());
IF HealthProbe.Health.TaskAvailable THEN
    PneumaticPress.SetSystemHealth(Input := HealthProbe.Health, ParCfg := HealthConfig);
ELSE
    ; // first monotonic sample has no prior scan from which to derive a period
END_IF

// First execute ordinary control, then apply a standard-PLC withdrawal layer.
// This is defense in depth only: the real safety system owns pneumatic removal.
PneumaticPress();
OutputAuthority.M_Apply(PressHal := PressHal, DoorHal := DoorHal,
    SlideHal := SlideHal, PowerFeedback := PowerHal.PowerFeedback,
    SafePneumaticPermit := SafePneumaticPermit,
    StandardIoHealthy := StandardIoHealthy,
    HazardousRamPermit := SafeGuardClosed AND SafeTwoHandActive);
IF USE_SIMULATION THEN
    // Never leave physical outputs energized while virtual commissioning.
    IoDriver.M_ClearOutputs();
    SimulationDriver.M_RefreshPlant();
ELSE
    LampsOn := PneumaticPress.OutImm.TwoHandStartReady;
    IoDriver.M_WriteOutputs(PressHal := PressHal, DoorHal := DoorHal,
        SlideHal := SlideHal, PowerHal := PowerHal, LampsOn := LampsOn,
        ControlCircuitMappingConfirmed := CONTROL_CIRCUIT_MAPPING_CONFIRMED,
        ForcePermitted := PneumaticPress.M_ForcePermitted());
END_IF
// Node state comes from the real EtherCAT master. §10.5.1 is a diagnostic
// surface, so the master is scanned only while a client is watching the bus
// view: the HMI sets FieldbusViewActive when its fieldbus page is open (the same
// on-demand gating the read tiers already apply to the topology data itself).
IoDriver.M_RefreshFieldbus(BusViewActive := FieldbusViewActive);

END_PROGRAM

// ---- 01_PneumaticPress/Recipes/FB_PressRecipeCatalog.TcPOU
// Owner-local recipe engineering data: model identities and their typed Unit records.
// Generic validation/storage remains in FB_LocalRecipeProvider; process behavior
// remains in the project-owned FB_PressDemoUnit. MAIN only composes the two.
FUNCTION_BLOCK FB_PressRecipeCatalog
VAR_OUTPUT
    {attribute 'OPC.UA.DA' := '0'}
    Provider : FB_LocalRecipeProvider;
END_VAR
VAR PERSISTENT
    // §3.8b - the records are edited through the Unit's model data (any model;
    // the provider's Save writes here) and must outlive a restart, so they are
    // retained and seeded only once.
    _default : ST_PneumaticPressParCfg;
    _aluminum : ST_PneumaticPressParCfg;
    _plastic : ST_PneumaticPressParCfg;
    _steel : ST_PneumaticPressParCfg;
    _seeded : UINT;               // RECIPE_SEED once the defaults below were written
END_VAR
VAR
    _model : ST_ModelId;
    _configured : BOOL;
END_VAR
VAR CONSTANT
    // Bump to re-seed every record with the design values below (a download that
    // changes them, or a record layout change).
    RECIPE_SEED : UINT := 1;
END_VAR

// Static catalog: no cyclic work.

METHOD Setup : BOOL
VAR_INPUT
    UnitRef : REFERENCE TO FB_PressDemoUnit;
END_VAR
VAR
    Ok : BOOL;
END_VAR
IF _configured THEN
    Setup := TRUE;
    RETURN;
END_IF

// §8.11 per-model performance references: IdealCycleMs feeds OEE Performance
// (§8.5.1); BaselineWorkMs arms the WORK-time degradation watch (§8.11.4(d)).
// Values = design cycle for this training cell (motions + settle + dwell).
// Seeded once: afterwards the retained records hold what was edited.
IF _seeded <> RECIPE_SEED THEN
    _default.PressSettleTime := T#500MS;
    _default.TransferSettleTime := T#100MS;
    _default.IdealCycleMs := 6000;
    _default.BaselineWorkMs := 6000;
    _aluminum.PressSettleTime := T#300MS;
    _aluminum.TransferSettleTime := T#80MS;
    _aluminum.IdealCycleMs := 5700;
    _aluminum.BaselineWorkMs := 5700;
    _plastic.PressSettleTime := T#650MS;
    _plastic.TransferSettleTime := T#120MS;
    _plastic.IdealCycleMs := 6200;
    _plastic.BaselineWorkMs := 6200;
    _steel.PressSettleTime := T#1200MS;
    _steel.TransferSettleTime := T#150MS;
    _steel.IdealCycleMs := 6800;
    _steel.BaselineWorkMs := 6800;
    _seeded := RECIPE_SEED;
END_IF

Ok := Provider.Register(ModelCode := '', RecipeKey := 'PneumaticPressUnit',
    pData := ADR(_default), Size := SIZEOF(_default));
Ok := Provider.Register(ModelCode := 'ALUMINUM', RecipeKey := 'PneumaticPressUnit',
    pData := ADR(_aluminum), Size := SIZEOF(_aluminum)) AND Ok;
Ok := Provider.Register(ModelCode := 'PLASTIC', RecipeKey := 'PneumaticPressUnit',
    pData := ADR(_plastic), Size := SIZEOF(_plastic)) AND Ok;
Ok := Provider.Register(ModelCode := 'STEEL', RecipeKey := 'PneumaticPressUnit',
    pData := ADR(_steel), Size := SIZEOF(_steel)) AND Ok;

_model.ModelCode := 'ALUMINUM';
Ok := UnitRef.RegisterAvailableModel(Id := _model) AND Ok;
_model.ModelCode := 'PLASTIC';
Ok := UnitRef.RegisterAvailableModel(Id := _model) AND Ok;
_model.ModelCode := 'STEEL';
Ok := UnitRef.RegisterAvailableModel(Id := _model) AND Ok;

_configured := Ok;
Setup := Ok;
END_METHOD

END_FUNCTION_BLOCK

// ---- 01_PneumaticPress/FB_PressDemoUnit.TcPOU
// Project-owned Unit: pneumatic press + access door + transfer slide + two-hand request.
// Cylinder interlocks prevent the two documented collisions in AUTO and MANUAL.
// Certified E-stop, two-hand evaluation and safe valve outputs remain external.
FUNCTION_BLOCK FB_PressDemoUnit EXTENDS FB_UnitBase
VAR_INPUT
    ParCfg : ST_PneumaticPressParCfg;
    ParCmd : ST_PneumaticPressParCmd;
END_VAR
VAR_OUTPUT
    PressRam      : FB_CylinderCM;
    Door          : FB_CylinderCM;
    PartSlide     : FB_CylinderCM;
    TwoHand       : FB_TwoHandStartCM;
    PneumaticPower: FB_PowerGroupCM;
    PartPresentSensor : FB_DigitalInputCM;
    AirPressureMonitor : FB_AirPressureMonitorCM;
    // Jenny Science XENAX Xvi servo (Annex G, PLCopen Motion). NOT CABINET
    // HARDWARE - read the note on PartFeedAxis before looking for it there.
    PartFeed      : FB_AxisCM;
    // Project-owned, browseable condition state of the rendition that RUNS.
    ReleaseConditions : ST_PressDemoReleaseConditions;
    OutCmd        : ST_PneumaticPressOutCmd;
    OutImm        : ST_PneumaticPressOutImm;
END_VAR
VAR
    {attribute 'OPC.UA.DA' := '0'}
    _recipe : I_RecipeProvider;
    // The NC axis this Unit feeds parts with. Until an axis is actually linked
    // in the System Manager, _partFeedConfigured stays FALSE and the module is
    // never called: MC_Power against an unlinked AXIS_REF would otherwise run
    // every scan on a bench whose eight tests are green. Absent hardware is
    // absent, not silently pretended.
    //
    // WHAT THIS AXIS IS, AND IS NOT (2026-08-25). The delivered CX2030 cabinet
    // has NO SERVO. Its approved I/O list is five Beckhoff terminals
    // (=000+S-K010: EK1200 / EL1809 / EL2809 / EL6001 / EL9011 -- see
    // Specification/Reports/CX2030_PRESS_IO_MAPPING.md), and the part feeder in
    // that cabinet is PNEUMATIC: PartSlide above, driven by the digital outputs
    // _101K301A/_101K301B. Do not go looking for this axis on the cabinet bus.
    //
    // The drive behind it is a Jenny Science XENAX Xvi (vendor #x557, product
    // #x7508) on a SECOND EtherCAT device, =000+S-A620 (EtherCAT), kept in its
    // own XTI beside the cabinet's. It is outside the press entirely and stands
    // in for a feed axis so a real process can be simulated against real motion
    // hardware. Anything it teaches (S3.8c) or persists (S3.8b) is BENCH data,
    // not commissioning data for the press -- which is why =000+S-A610-A1
    // (EtherCAT).xti, the faithful record of the delivered cabinet, does not
    // mention it and must not be made to.
    {attribute 'OPC.UA.DA' := '0'}
    PartFeedAxis : AXIS_REF;
    _partFeedConfigured : BOOL;
    _partFeedArmed : BOOL;             // last arming attempt's result (S5.6: no discarded return)
    // §10.5.1 - the project I/O catalog owns the approved channel identity join
    // (§10.2.1), so it, not this Unit, resolves a force request to a physical
    // channel. Absent = no force routing, which is the fail-closed default.
    {attribute 'OPC.UA.DA' := '0'}
    _ioCatalog : REFERENCE TO FB_PressIoCatalog;
    _parCfgStaged : ST_PneumaticPressParCfg;
    // §3.8a - the ParCfg last applied (commit or accepted edit); a difference is an
    // edit of the active model's recipe to take effect and to write back.
    {attribute 'OPC.UA.DA' := '0'}
    _parCfgApplied : ST_PneumaticPressParCfg;
    _recipePrepared : BOOL;
    _startLatched : BOOL;
    _powerRequestPending : BOOL;
    _powerTargetOn : BOOL;
    {attribute 'OPC.UA.DA' := '0'}
    _homeSequence : FB_PressDemoHome;       // §6.8 ST chain on FB_SequenceBase owns HOME steps
    {attribute 'OPC.UA.DA' := '0'}
    _changeoverSequence : FB_PressDemoChangeover;
    // §6.8 / O2 — the SAME AUTO chain in all three permitted languages. This is a
    // demo bench: carrying three renditions is the point (O2 says sequences and
    // interlocks may be ST, SFC or Ladder), not something a real project would do.
    // AUTO_SEQUENCE_LANGUAGE below picks which one the Unit binds and runs; the
    // other two are inert. They are excluded from OPC UA for the same reason the
    // bound one is: a chain is not a module and publishes no Status.
    {attribute 'OPC.UA.DA' := '0'}
    _autoSequence : FB_PressDemoAuto;
    {attribute 'OPC.UA.DA' := '0'}
    _sfcAutoSequence : FB_SFC_PressDemoAuto;
    {attribute 'OPC.UA.DA' := '0'}
    _ldAutoSequence : FB_LD_PressDemoAuto;
    // §7.2 / O2 — the SAME release engineering in a second language. Only the
    // rendition RELEASE_LANGUAGE selects is set up, evaluated, and allowed to
    // write the directional permits and the release report; the other is inert.
    // Neither rendition is published itself: the selected one fills
    // ReleaseConditions (a VAR_OUTPUT above) every scan, so the browseable
    // record is always the one being evaluated. Publishing the ST instance
    // directly left it frozen at FALSE whenever LD was selected (§3.12).
    {attribute 'OPC.UA.DA' := '0'}
    _stReleaseConditions : FB_PressDemoRelease;
    {attribute 'OPC.UA.DA' := '0'}
    _ldReleaseConditions : FB_LD_PressDemoRelease;
END_VAR
VAR PERSISTENT
    // §3.8b - this station's deployment data. PERSISTENT is the BACKING, not the
    // architecture: the values are reached as (Scope, WriteKey) capabilities like
    // every other editable value, never as an aggregate copied in and out.
    _station : ST_PneumaticPressStationCfg;
END_VAR
VAR CONSTANT
    // §3.8b - layout version of the retained image above. Bump it when a member
    // is added, and the old image is rejected and annunciated instead of read by
    // field position.
    PRESS_STATIONCFG_SCHEMA : UINT := 1;
    // §3.8 - the longest settle times a recipe may hold. ONE source for the check
    // a changeover applies (PrepareRecipe) and the range an edit is offered
    // (the PAR_CFG registration), so an edit can never store what a changeover
    // would refuse.
    RECIPE_MAX_PRESS_SETTLE_MS    : UDINT := 30000;
    RECIPE_MAX_TRANSFER_SETTLE_MS : UDINT := 5000;
    // The provider key of this Unit's recipe record: loaded at a changeover and
    // edited per model through the same key (§3.8a).
    PRESS_RECIPE_KEY : STRING(80) := 'PneumaticPressUnit';
    // Which rendition of the AUTO chain runs. VAR CONSTANT on purpose, like the
    // §6.0 commissioning gates in MAIN: switching language is a source edit plus a
    // download, never an online write. The compiler folds the unselected branches.
    //   STRUCTURED_TEXT           -> FB_PressDemoAuto
    //   SEQUENTIAL_FUNCTION_CHART -> FB_SFC_PressDemoAuto
    //   LADDER_DIAGRAM            -> FB_LD_PressDemoAuto
    AUTO_SEQUENCE_LANGUAGE : E_RenditionLanguage := E_RenditionLanguage.LADDER_DIAGRAM;
    // Which rendition of the release/interlock logic is evaluated, on the same
    // terms and from the same type, so a value means the same language in both
    // selections. There is no SEQUENTIAL_FUNCTION_CHART rendition here: SFC is a
    // sequence language and has nothing to say about a permissive, so that
    // member is simply never selected rather than being given a second meaning.
    //   STRUCTURED_TEXT -> FB_PressDemoRelease
    //   LADDER_DIAGRAM  -> FB_LD_PressDemoRelease
    RELEASE_LANGUAGE : E_RenditionLanguage := E_RenditionLanguage.LADDER_DIAGRAM;
END_VAR

Cyclic();

// §7.8 mode-entry release owned by this Unit. The base Start method consumes the
// same report the HMI displays, so this condition cannot become explanation-only.
METHOD PROTECTED _M_AppendInterlocks
VAR_IN_OUT
    Report : ST_ReleaseReport;
END_VAR
IF ModeActive <> E_Mode.CHANGEOVER THEN
IF RELEASE_LANGUAGE = E_RenditionLanguage.LADDER_DIAGRAM THEN
    _ldReleaseConditions.M_AppendStart(Report := Report);
ELSE
    _stReleaseConditions.M_AppendStart(Report := Report);
END_IF
END_IF
END_METHOD

METHOD PROTECTED _M_AppendManualInterlocks
VAR_INPUT
    TargetPath : STRING(255);
    Value : DINT;
END_VAR
VAR_IN_OUT
    Report : ST_ReleaseReport;
END_VAR
IF RELEASE_LANGUAGE = E_RenditionLanguage.LADDER_DIAGRAM THEN
    _ldReleaseConditions.M_AppendManual(TargetPath := TargetPath, Value := Value,
        PressRam := PressRam, Door := Door, PartSlide := PartSlide, Report := Report);
ELSE
    _stReleaseConditions.M_AppendManual(TargetPath := TargetPath, Value := Value,
        PressRam := PressRam, Door := Door, PartSlide := PartSlide, Report := Report);
END_IF
END_METHOD

// Clear state that must not survive init, mode entry, or either abort path. The
// base already restarts the chains and clears their decision (§6.8); this is the
// Unit's OWN state. OnCommandStart deliberately does not call this: a physical
// start pulse may have been latched one scan before the Execute edge is consumed.
METHOD PROTECTED _M_ClearModeTransitionState
_startLatched := FALSE;
END_METHOD

// Thin mode router. Each supported sequence is a named method in the Unit tree.
METHOD PROTECTED _M_Dispatch
CASE ModeActive OF
    E_Mode.AUTO:
        _M_SequenceAuto();
    E_Mode.HOME:
        _M_SequenceHome();
    E_Mode.CHANGEOVER:
        _M_SequenceChangeover();
    E_Mode.MANUAL:
        _M_Fault(E_Reason.UNSUPPORTED_COMMAND, 'project.error.pressManualHasNoSequence');
ELSE
    _M_Fault(E_Reason.UNSUPPORTED_COMMAND, 'project.error.pressModeHasNoSequence');
END_CASE
END_METHOD

// §10.2.1 — inject this station's I/O catalog so §10.5.1 force requests can be
// resolved against the approved engineering-data join instead of against a
// second copy of the channel map. Wired once by the composition root.
METHOD SetIoCatalog
VAR_INPUT
    Catalog : REFERENCE TO FB_PressIoCatalog;
END_VAR
_ioCatalog REF= Catalog;
END_METHOD

// §10.5.1 — resolve an accepted force request onto a physical output channel.
// FB_UnitBase.ForceChannel has already proved the §7.7 MANUAL access level, the
// §7.5 OUTPUT_FORCING build gate, and that this Unit is idle in MANUAL; the
// catalog then proves what only it knows — that the path names a channel of THIS
// root, that it is an OUTPUT, and that the project marked it forceable.
METHOD PROTECTED _M_RouteForceChannel : BOOL
VAR_INPUT
    ChannelPath : STRING(255);
    Force       : BOOL;
    BoolText    : STRING(255);
    AnalogText  : STRING(160);
END_VAR
_M_RouteForceChannel := FALSE;
IF NOT __ISVALIDREF(_ioCatalog) THEN
    RETURN;
END_IF
// The transported value is text (the mailbox carries no variant), so a malformed
// payload must decode to a defined value rather than to whatever the converter
// leaves behind: anything that is not exactly 'true' is FALSE (§5.6).
_M_RouteForceChannel := _ioCatalog.M_RouteForce(ChannelPath := ChannelPath,
    OwnerRootPath := _name, Force := Force,
    BoolValue := (BoolText = 'true'),
    AnalogValue := STRING_TO_REAL(AnalogText));
END_METHOD

// Wiring-only AUTO adapter. Every production command, wait, timer, decision,
// traceability action, and transition lives in the §6.8 chain.
METHOD PROTECTED _M_SequenceAuto
// An ST chain's body is a method (M_Run); an SFC or LD chain's body IS the chart,
// so the instance itself is the call. That asymmetry is the language difference,
// not an inconsistency to normalise away.
IF AUTO_SEQUENCE_LANGUAGE = E_RenditionLanguage.LADDER_DIAGRAM THEN
    _ldAutoSequence();
ELSIF AUTO_SEQUENCE_LANGUAGE = E_RenditionLanguage.SEQUENTIAL_FUNCTION_CHART THEN
    _sfcAutoSequence();
ELSE
    _autoSequence.M_Run();
END_IF
END_METHOD

// Wiring-only CHANGEOVER adapter. The §6.8 chain owns model validation, safe
// positioning, the operator decision, and completion logic.
METHOD PROTECTED _M_SequenceChangeover
_changeoverSequence.M_Run();
END_METHOD

// Wiring-only HOME adapter. OnCommandStart owns the reset edge; the sequence POU
// owns every process step and terminal action.
METHOD PROTECTED _M_SequenceHome
_homeSequence.M_Run();
END_METHOD

METHOD PROTECTED _M_Supports : BOOL
VAR_INPUT
    Mode : E_Mode;
END_VAR
_M_Supports := (Mode = E_Mode.AUTO) OR (Mode = E_Mode.MANUAL)
    OR (Mode = E_Mode.HOME) OR (Mode = E_Mode.CHANGEOVER);
END_METHOD

// §3.4.2 — the press paces every motion boundary through _M_StepGate, so
// SINGLE_STEP and HOLD_TO_RUN are supported (NON-SAFETY pacing; interlocks
// and the certified safety layer are unaffected).
METHOD PROTECTED _M_SupportsRunStyle : BOOL
VAR_INPUT
    Style : E_RunStyle;
END_VAR
_M_SupportsRunStyle := (Style = E_RunStyle.CONTINUOUS)
    OR (Style = E_RunStyle.SINGLE_STEP) OR (Style = E_RunStyle.HOLD_TO_RUN);
END_METHOD

// One safe-stop wiring point shared by normal and error-state abort transitions.
METHOD PROTECTED _M_WithdrawSequenceOutputs
PressRam.WithdrawOutputs();
Door.WithdrawOutputs();
PartSlide.WithdrawOutputs();
PressRam.Execute := FALSE;
Door.Execute := FALSE;
PartSlide.Execute := FALSE;
END_METHOD

METHOD AbortRecipe
SUPER^.AbortRecipe();
_recipePrepared := FALSE;
END_METHOD

METHOD CommitRecipe
SUPER^.CommitRecipe();
IF _recipePrepared THEN
    ParCfg := _parCfgStaged;
    // §8.11 performance references follow the model: OEE Performance denominator
    // and the WORK-time degradation baseline are per-recipe engineering data.
    Oee.IdealCycleMs := ParCfg.IdealCycleMs;
    Profiler.M_SetBaselineWork(WorkMs := ParCfg.BaselineWorkMs);
    _parCfgApplied := ParCfg;
END_IF
_recipePrepared := FALSE;
END_METHOD

// §3.10.2 — base walk (Unit facets + all child modules), then the project-owned
// fieldbus topology identity, from the I/O catalog that owns it (SetIoCatalog):
// its static members are OPC.UA.DA=0 and reach the HMI only through this manifest.
METHOD M_AppendConfig : BOOL
VAR_INPUT
    Pager : REFERENCE TO FB_ConfigPager;
END_VAR
M_AppendConfig := SUPER^.M_AppendConfig(Pager := Pager);
IF __ISVALIDREF(_ioCatalog) THEN
    _ioCatalog.M_AppendTopologyConfig(Pager := Pager);
END_IF
END_METHOD

METHOD PROTECTED OnAbort : DINT
OnAbort := SUPER^.OnAbort();
_M_PartAborted();                    // §3.16.3: the part leaves without a valid result
_M_WithdrawSequenceOutputs();
_M_ClearModeTransitionState();
_powerTargetOn := FALSE;
_powerRequestPending := TRUE;
END_METHOD

// Error-state Abort is a deliberate recovery action but does not clear ERROR.
METHOD PROTECTED OnAbortInError : DINT
OnAbortInError := SUPER^.OnAbortInError();
_M_WithdrawSequenceOutputs();
_M_ClearModeTransitionState();
_powerTargetOn := FALSE;
_powerRequestPending := TRUE;
END_METHOD

// The press's restart policy (§6.9(d)): every accepted Start gets a fresh mode
// chain, including a repeated HOME/CHANGEOVER run that does not pass through
// another mode change. Resuming where an error stopped is the other legitimate
// choice; this station does not make it.
METHOD PROTECTED OnCommandStart : DINT
OnCommandStart := SUPER^.OnCommandStart();
_M_RestartSequences();
END_METHOD

METHOD PROTECTED OnCyclic : DINT
VAR
    started : BOOL;
END_VAR
OnCyclic := SUPER^.OnCyclic();
// §3.8b/§3.12 — the step guard is DERIVED from the station value every scan, not
// latched at Setup. An operator who edits press.stallGuardMs gets the new guard
// on the next step, and the published StallTime can never disagree with the
// configuration it came from.
StallTime := UDINT_TO_TIME(_station.StallGuardMs);
// §3.8a - an accepted edit of the ACTIVE model's recipe lands in ParCfg (the base
// has already saved it to the model's record). The performance references follow
// it, as they do at a changeover.
IF MEMCMP(ADR(ParCfg), ADR(_parCfgApplied), SIZEOF(ParCfg)) <> 0 THEN
    Oee.IdealCycleMs := ParCfg.IdealCycleMs;
    Profiler.M_SetBaselineWork(WorkMs := ParCfg.BaselineWorkMs);
    _parCfgApplied := ParCfg;
END_IF
// §7.2.1/§6.1 - a cylinder cannot move without air, so air is each cylinder's own
// process condition. Lost mid-stroke, the cylinder HOLDS - outputs off, resumes by
// itself when pressure returns - and the Unit rolls the hold up by name. Nothing
// to reset: the process restores this condition, it is not a defect.
PressRam.SetAreaSafe(Ok := AirPressureMonitor.OutImm.PressureOk,
    DescriptionKey := 'project.interlock.pressRequiresAirPressure');
Door.SetAreaSafe(Ok := AirPressureMonitor.OutImm.PressureOk,
    DescriptionKey := 'project.interlock.pressRequiresAirPressure');
PartSlide.SetAreaSafe(Ok := AirPressureMonitor.OutImm.PressureOk,
    DescriptionKey := 'project.interlock.pressRequiresAirPressure');
// Project release engineering is a separate visible component. It owns the
// functional collision permits and mode-entry conditions consumed below.
IF RELEASE_LANGUAGE = E_RenditionLanguage.LADDER_DIAGRAM THEN
    _ldReleaseConditions.M_Evaluate(PressRam := PressRam, Door := Door, PartSlide := PartSlide,
        TwoHand := TwoHand, PneumaticPower := PneumaticPower,
        AirPressure := AirPressureMonitor);
    _ldReleaseConditions.M_PublishTo(Conditions := ReleaseConditions);
ELSE
    _stReleaseConditions.M_Evaluate(PressRam := PressRam, Door := Door, PartSlide := PartSlide,
        TwoHand := TwoHand, PneumaticPower := PneumaticPower,
        AirPressure := AirPressureMonitor);
    _stReleaseConditions.M_PublishTo(Conditions := ReleaseConditions);
END_IF

// S1.1 O1 - the axis ARMS ITSELF on the first scan a real NC axis is behind
// it, rather than through a call a composition root has to remember. Forgetting
// such a call produces a silently dead module, which is exactly the class of
// defect the objective says to drive from a path the application already takes.
// ConfigurePartFeedAxis is idempotent and fails closed, so calling it until it
// succeeds costs one comparison per scan on a bench with no drive.
IF NOT _partFeedConfigured THEN
    // THIS^ is required: an unqualified same-FB call resolves only when its
    // return value is discarded, and this one is not (C0009/C0035 otherwise).
    _partFeedArmed := THIS^.ConfigurePartFeedAxis(AxisRef := PartFeedAxis);
END_IF
// The feed axis runs only once an NC axis has been linked (S10.6). Its
// conditions are re-driven every scan so a manual move obeys the same rule as
// a sequenced one (S7.2).
//
// The module itself is NOT called here: ConfigurePartFeedAxis registers it as a
// child, and _M_TickChildren already ticks every registered child from
// SUPER^.OnCyclic above. Calling it here as well would run the whole S6.1
// lifecycle twice per scan.
// No conditions are driven here any more. Both that used to be - the press's
// pneumatic power and its ram guard - describe the PRESS, and the Xvi is
// physically outside it on a separate EtherCAT device. Gating a bench servo on
// whether a pneumatic valve zone somewhere else is energised is not an
// interlock, it is an unrelated fact that happens to block motion, and S7.2.1
// says a condition is defined at the module with enough semantic context to own
// it. This Unit has none for that drive.

// Latch access-gated Unit requests, then observe one full Execute-low scan before
// starting another power-group command (PLCopen edge discipline).
IF ControlOffRequest THEN
    _powerTargetOn := FALSE;
    _powerRequestPending := TRUE;
ELSIF ControlOnRequest THEN
    _powerTargetOn := TRUE;
    _powerRequestPending := TRUE;
END_IF
IF PneumaticPower.Done OR PneumaticPower.Error OR PneumaticPower.Aborted THEN
    PneumaticPower.Execute := FALSE;
ELSIF _powerRequestPending AND NOT PneumaticPower.Execute
AND (PneumaticPower.State = E_ExecState.READY) THEN
    PneumaticPower.Abort := FALSE;
    IF _powerTargetOn THEN
        PneumaticPower.Command := E_PowerGroupCommand.POWER_ON;
    ELSE
        PneumaticPower.Command := E_PowerGroupCommand.POWER_OFF;
    END_IF
    PneumaticPower.Execute := TRUE;
    _powerRequestPending := FALSE;
END_IF

// A physical two-hand edge starts AUTO from READY, or releases a running Unit's
// two-hand wait. Start() is asked unconditionally: its release report is the whole
// start predicate and names whatever refuses it (§7.2.1, §7.8). What IS qualified
// is the start LATCH: a press counts only when the part and the air that the N100
// wait also names are already there, so a press made before the part was loaded
// can never start the stroke when the part arrives. N100 shows what it waits for.
IF TwoHand.OutImm.StartPulse THEN
    IF ModeActive = E_Mode.AUTO THEN
        IF State = E_ExecState.BUSY THEN
            started := TRUE;
        ELSE
            started := Start();
        END_IF
        _startLatched := started
            AND PartPresentSensor.OutImm.Value AND PartPresentSensor.OutImm.Quality
            AND AirPressureMonitor.OutImm.PressureOk;
    ELSE
        _startLatched := FALSE;
    END_IF
END_IF
IF PneumaticPower.Error AND (State = E_ExecState.BUSY) THEN
    _M_RollupFault();
END_IF
// §3.12 — ONE derivation, published under the name the operator knows and read
// by everything that needs the fact (§1.1 O9: derived, never duplicated). It is a
// state, not a command result: it stops being true the moment a cylinder leaves
// the position, including in MANUAL where no sequence runs to clear anything.
// _M_State publishes it on the generic flag table with the moment it last changed,
// so the HMI can render it without knowing this module type.
OutImm.Homed := _M_State(Idx := 1, Key := 'project.state.pressAtLoadPosition',
    Ok := Door.OutImm.Retracted AND NOT Door.OutImm.Extended
      AND PartSlide.OutImm.Retracted AND NOT PartSlide.OutImm.Extended
      AND PressRam.OutImm.Retracted AND NOT PressRam.OutImm.Extended);
// The pushbutton lamps' condition, derived here - where the facts live - so the
// composition root only maps it to the output (§10.2.1).
OutImm.TwoHandStartReady := _M_State(Idx := 2, Key := 'project.state.pressTwoHandStartReady',
    Ok := TwoHand.OutImm.Armed AND ControlDomain.ReadyForStart
      AND PartPresentSensor.OutImm.Value AND PartPresentSensor.OutImm.Quality
      AND AirPressureMonitor.OutImm.PressureOk);
END_METHOD

// First operational scan: initialize application-owned mode-chain state.
METHOD PROTECTED OnInit : DINT
OnInit := SUPER^.OnInit();
_M_ClearModeTransitionState();
END_METHOD

// Mode-entry wiring only. Step behavior remains in the selected sequence POU.
METHOD PROTECTED OnModeChanged : DINT
VAR_INPUT
    NewMode : E_Mode;
    OldMode : E_Mode;
END_VAR
OnModeChanged := SUPER^.OnModeChanged(
    NewMode := NewMode, OldMode := OldMode);
_M_ClearModeTransitionState();
END_METHOD

// An operator reset is recovering this Unit: put the application back to the same
// safe wiring an error-state abort establishes, so the reset the operator presses at
// the panel needs no separate Stop/Abort first. The base then releases the run
// command and the children's commands, so the next HOME gets a genuine command edge.
// Unlike the abort paths this does NOT touch control power in either direction: it
// never requests Control On (§9.8 forbids self-resume), and it must not request
// Control Off either — powering down a healthy control circuit would make the
// operator re-enable it before HOME could run, i.e. reintroduce the multi-action
// recovery this reset exists to remove. Power stays where the operator put it.
METHOD PROTECTED OnOperatorReset : DINT
OnOperatorReset := SUPER^.OnOperatorReset();
_M_WithdrawSequenceOutputs();
_M_RestartSequences();                // this station restarts after a reset (§6.9(d))
_M_ClearModeTransitionState();
END_METHOD

METHOD PrepareRecipe : BOOL
VAR_INPUT
    Model : ST_ModelId;
END_VAR
IF _recipe = 0 THEN
    _parCfgStaged := ParCfg;
    _recipePrepared := TRUE;
ELSIF _recipe.Load(ModelCode := Model.ModelCode, RecipeKey := PRESS_RECIPE_KEY, pParCfg := ADR(_parCfgStaged), Size := SIZEOF(_parCfgStaged)) THEN
    IF (TIME_TO_UDINT(_parCfgStaged.PressSettleTime) > RECIPE_MAX_PRESS_SETTLE_MS)
    OR (TIME_TO_UDINT(_parCfgStaged.TransferSettleTime) > RECIPE_MAX_TRANSFER_SETTLE_MS) THEN
        _M_Fault(E_Reason.RECIPE_INVALID, 'project.error.pressRecipeInvalid');
        _recipePrepared := FALSE;
        PrepareRecipe := FALSE;
        RETURN;
    END_IF
    _recipePrepared := TRUE;
ELSE
    _M_Fault(E_Reason.RECIPE_INVALID, 'std.error.recipeSchemaInvalid');
    _recipePrepared := FALSE;
    PrepareRecipe := FALSE;
    RETURN;
END_IF
PrepareRecipe := SUPER^.PrepareRecipe(Model := Model);
IF NOT PrepareRecipe THEN _recipePrepared := FALSE; END_IF
END_METHOD

// Application-only seam for ordinary hardwired Control On/Off buttons.
// It is a method (not OPC UA data), so HMI writes still use the access-gated
// ReqControlOn/ReqControlOff contract. The power CM rechecks safety and health.
METHOD RequestLocalControl : BOOL
VAR_INPUT
    ControlOn : BOOL;
END_VAR
_powerTargetOn := ControlOn;
_powerRequestPending := TRUE;
RequestLocalControl := TRUE;
END_METHOD

METHOD Setup : BOOL
VAR_INPUT
    Name : STRING(80);
    PressHal : REFERENCE TO ST_CylinderHal;
    DoorHal : REFERENCE TO ST_CylinderHal;
    SlideHal : REFERENCE TO ST_CylinderHal;
    TwoHandHal : REFERENCE TO ST_TwoHandHal;
    PowerHal : REFERENCE TO ST_PowerGroupHal;
    PartPresentHal : REFERENCE TO ST_DigitalInputHal;
    AirPressureHal : REFERENCE TO ST_AirPressureHal;
    Recipe : I_RecipeProvider;
END_VAR
VAR
    InitialModel : ST_ModelId;
    Ok : BOOL;
END_VAR
_M_SetName(Name);
_M_SetPresentation(DisplayNameKey := 'project.module.pneumaticPress.name', DescriptionKey := 'project.module.pneumaticPress.description', TypeKey := 'project.moduleType.pneumaticPress');
_recipe := Recipe;
Ok := PressRam.Setup(Name := CONCAT(Name, '.PressRam'), HalRef := PressHal, Recipe := 0);
Ok := Door.Setup(Name := CONCAT(Name, '.Door'), HalRef := DoorHal, Recipe := 0) AND Ok;
Ok := PartSlide.Setup(Name := CONCAT(Name, '.PartSlide'), HalRef := SlideHal, Recipe := 0) AND Ok;
Ok := TwoHand.Setup(Name := CONCAT(Name, '.TwoHand'), HalRef := TwoHandHal) AND Ok;
Ok := PneumaticPower.Setup(Name := CONCAT(Name, '.PneumaticPower'), HalRef := PowerHal) AND Ok;
Ok := PartPresentSensor.Setup(Name := CONCAT(Name, '.PartPresentSensor'),
    HalRef := PartPresentHal, DisplayNameKey := 'project.module.partPresentSensor.name',
    DescriptionKey := 'project.module.partPresentSensor.description') AND Ok;
Ok := AirPressureMonitor.Setup(Name := CONCAT(Name, '.AirPressureMonitor'),
    HalRef := AirPressureHal) AND Ok;
IF RELEASE_LANGUAGE = E_RenditionLanguage.LADDER_DIAGRAM THEN
    Ok := _ldReleaseConditions.Setup(UnitPath := Name) AND Ok;
ELSE
    Ok := _stReleaseConditions.Setup(UnitPath := Name) AND Ok;
END_IF
Ok := _homeSequence.Setup(Host := THIS^, PressRam := PressRam, Door := Door,
    PartSlide := PartSlide, OutCmd := OutCmd) AND Ok;
Ok := _changeoverSequence.Setup(Host := THIS^, PressRam := PressRam, Door := Door,
    PartSlide := PartSlide, OutCmd := OutCmd, Model := Model) AND Ok;
// Only the selected rendition is attached: M_Attach registers the chain with the
// Unit, so attaching all three would put three chains on one step pointer.
// §3.8b restore, BEFORE the chains are set up: they take _station by reference
// and the first scan must already see either the commissioned values or the
// declared defaults, never a half-initialized image. The rule itself lives in
// FB_ModuleBase - this type supplies only what is genuinely its own, which is
// what its defaults are.
IF NOT M_RestoreStationCfg(pVersion := ADR(_station.SchemaVersion),
        SchemaVersion := PRESS_STATIONCFG_SCHEMA) THEN
    // Fail-safe defaults: two-hand REQUIRED (a lost risk-assessment policy must
    // never come back as the permissive one), and the framework's own 30 s
    // stall guard.
    _station.RequireTwoHandStart := TRUE;
    _station.StallGuardMs := 30000;
END_IF
IF AUTO_SEQUENCE_LANGUAGE = E_RenditionLanguage.LADDER_DIAGRAM THEN
    Ok := _ldAutoSequence.Setup(Host := THIS^, PressRam := PressRam, Door := Door,
        PartSlide := PartSlide, TwoHand := TwoHand, PartPresentSensor := PartPresentSensor,
        AirPressureMonitor := AirPressureMonitor, ParCfg := ParCfg,
        StationCfg := _station, OutCmd := OutCmd,
        StartLatched := _startLatched) AND Ok;
ELSIF AUTO_SEQUENCE_LANGUAGE = E_RenditionLanguage.SEQUENTIAL_FUNCTION_CHART THEN
    Ok := _sfcAutoSequence.Setup(Host := THIS^, PressRam := PressRam, Door := Door,
        PartSlide := PartSlide, TwoHand := TwoHand, PartPresentSensor := PartPresentSensor,
        AirPressureMonitor := AirPressureMonitor, ParCfg := ParCfg,
        StationCfg := _station, OutCmd := OutCmd,
        StartLatched := _startLatched) AND Ok;
ELSE
    Ok := _autoSequence.Setup(Host := THIS^, PressRam := PressRam, Door := Door,
        PartSlide := PartSlide, TwoHand := TwoHand, PartPresentSensor := PartPresentSensor,
        AirPressureMonitor := AirPressureMonitor, ParCfg := ParCfg,
        StationCfg := _station, OutCmd := OutCmd,
        StartLatched := _startLatched) AND Ok;
END_IF
PneumaticPower.ParCfg.Kind := E_PowerGroupKind.VALVE_ZONE;
PneumaticPower.ParCfg.RequiredForControl := TRUE;
PneumaticPower.ParCfg.FieldbusLossReaction := E_FieldbusLossReaction.CONTROL_OFF;
Ok := _M_Register(PressRam) AND Ok;
Ok := _M_Register(Door) AND Ok;
Ok := _M_Register(PartSlide) AND Ok;
Ok := _M_Register(TwoHand) AND Ok;
Ok := _M_Register(PneumaticPower) AND Ok;
Ok := _M_Register(PartPresentSensor) AND Ok;
Ok := _M_Register(AirPressureMonitor) AND Ok;
// §3.8a/§3.10.2 - the two deployment values become editable CAPABILITIES. That
// registration, not publication and not DATA_WRITE, is what makes them writable,
// and it is also what puts them into a station parameter set: SaveConfigSet walks
// the same registry (§3.8b), so a value registered here needs no separate line
// anywhere to be saved, listed, exported and restored.
Ok := M_RegisterConfigFlag(Key := 'press.requireTwoHandStart',
    Item := 'StationCfg/RequireTwoHandStart',
    LabelKey := 'project.config.pressRequireTwoHandStart',
    Kind := E_ConfigKind.STATION_CFG, pTarget := ADR(_station.RequireTwoHandStart),
    RequiresReady := TRUE) AND Ok;
Ok := M_RegisterConfigNumber(Key := 'press.stallGuardMs',
    Item := 'StationCfg/StallGuardMs',
    LabelKey := 'project.config.pressStallGuardMs', Unit := E_EngUnit.MILLISECOND,
    Kind := E_ConfigKind.STATION_CFG, Storage := E_ConfigStorage.AS_UDINT,
    pTarget := ADR(_station.StallGuardMs), Minimum := 1000.0, Maximum := 600000.0,
    RequiresReady := TRUE) AND Ok;
// §3.8a - model data, PAR_CFG, over this Unit's recipe record. Registering the
// record makes these values editable for EVERY model in the catalog, and the base
// writes each edit back to that model's record. The ranges are the RECIPE_MAX_*
// constants PrepareRecipe also enforces.
IF Recipe <> 0 THEN
    Ok := M_RegisterModelData(pData := ADR(ParCfg), Size := SIZEOF(ParCfg),
        RecipeKey := PRESS_RECIPE_KEY, Provider := Recipe) AND Ok;
END_IF
Ok := M_RegisterConfigDuration(Key := 'press.recipe.pressSettle',
    Item := 'ParCfg/PressSettleTime', LabelKey := 'project.config.pressSettleTime',
    Kind := E_ConfigKind.PAR_CFG, pTarget := ADR(ParCfg.PressSettleTime),
    MinimumMs := 0, MaximumMs := RECIPE_MAX_PRESS_SETTLE_MS, RequiresReady := TRUE) AND Ok;
Ok := M_RegisterConfigDuration(Key := 'press.recipe.transferSettle',
    Item := 'ParCfg/TransferSettleTime', LabelKey := 'project.config.transferSettleTime',
    Kind := E_ConfigKind.PAR_CFG, pTarget := ADR(ParCfg.TransferSettleTime),
    MinimumMs := 0, MaximumMs := RECIPE_MAX_TRANSFER_SETTLE_MS, RequiresReady := TRUE) AND Ok;
Ok := M_RegisterConfigNumber(Key := 'press.recipe.idealCycleMs',
    Item := 'ParCfg/IdealCycleMs', LabelKey := 'project.config.idealCycleMs',
    Unit := E_EngUnit.MILLISECOND, Kind := E_ConfigKind.PAR_CFG,
    Storage := E_ConfigStorage.AS_UDINT, pTarget := ADR(ParCfg.IdealCycleMs),
    Minimum := 0.0, Maximum := 600000.0, RequiresReady := TRUE) AND Ok;
Ok := M_RegisterConfigNumber(Key := 'press.recipe.baselineWorkMs',
    Item := 'ParCfg/BaselineWorkMs', LabelKey := 'project.config.baselineWorkMs',
    Unit := E_EngUnit.MILLISECOND, Kind := E_ConfigKind.PAR_CFG,
    Storage := E_ConfigStorage.AS_UDINT, pTarget := ADR(ParCfg.BaselineWorkMs),
    Minimum := 0.0, Maximum := 600000.0, RequiresReady := TRUE) AND Ok;
Setup := Ok AND PrepareRecipe(Model := InitialModel);
IF Setup THEN CommitRecipe(); END_IF
END_METHOD

// Bind the NC axis for the part-feed servo and arm the module.
//
// Called from OnCyclic until it succeeds, so the axis arms itself the moment an
// NC axis is linked and stays dormant forever on a bench without one. It is
// idempotent and fails closed on both an invalid reference and an unlinked one
// (AxisId 0), which is what makes calling it every scan safe.
//
// The drive is a Jenny Science XENAX Xvi over EtherCAT/CiA402 on the DEV PC's
// own bus - a stand-in for a feed axis, not press cabinet hardware. See the
// note on PartFeedAxis.
//
// The conditions are declared HERE rather than in FB_PressDemoRelease only
// because the axis is not yet in the AUTO chain. When it joins the chain they
// belong beside the other project permits in the Release object, which S7.2.1
// prefers as a single visible component, and this method should shrink to
// binding the reference.
//
// ParCfg limits are deliberately NOT set here. Soft limits, velocity and
// acceleration come from the axis configuration and the recipe (S10.3); a Unit
// that hard-codes a stroke is wrong the first time the mechanics change.
METHOD ConfigurePartFeedAxis : BOOL
VAR_INPUT
    AxisRef : REFERENCE TO AXIS_REF;
END_VAR
IF NOT __ISVALIDREF(AxisRef) THEN
    ConfigurePartFeedAxis := FALSE;
    RETURN;
END_IF
// An AXIS_REF the System Manager has not linked to an NC axis carries AxisId 0.
// This is the test that keeps "absent hardware is absent" true now that arming
// is automatic: without it, a bench with no drive would Setup the module and
// start commanding MC_Power against nothing.
IF AxisRef.NcToPlc.AxisId = 0 THEN
    ConfigurePartFeedAxis := FALSE;
    RETURN;
END_IF
ConfigurePartFeedAxis := PartFeed.Setup(Name := CONCAT(Name, '.PartFeed'),
    AxisRef := AxisRef, Recipe := 0);
IF NOT ConfigurePartFeedAxis THEN
    RETURN;
END_IF
// No project conditions are declared for this axis, and the absence is the
// point rather than an omission. The two that used to be here required the
// press's pneumatic power and its ram guard to be satisfied before the axis
// could move - but the Xvi sits on =000+S-A620, a separate EtherCAT device
// outside the press, with its own power. Neither fact says anything about
// whether that drive may move.
//
// Declaring a condition that does not describe the device is worse than
// declaring none: it blocks motion for a reason the operator cannot act on, and
// it puts a name in the release report that is simply not about this axis
// (S7.2.1 - a condition belongs to the module with the semantic context to own
// it). If this drive is ever mounted INTO a cell, its real conditions get
// declared here then, from that cell's guard and power.
//
// The device-intrinsic gates are untouched and still apply: the axis will not
// jog stale, will not jog while a command owns it, and will not jog without a
// linked NC axis (FB_AxisCM._M_JogCyclic).
// Registered only once it is REAL. A registered child is ticked every scan,
// joins the S8.2 first-out rollup, and appears in the S3.10.2 config walk - and
// therefore in station parameter sets (S3.8b). Registering it unconditionally at
// Setup would put an unnamed module in the published tree and a taught position
// in every saved set for hardware that is not there.
ConfigurePartFeedAxis := _M_Register(PartFeed);
IF NOT ConfigurePartFeedAxis THEN
    RETURN;                            // no free child slot: stay dormant
END_IF
_partFeedConfigured := TRUE;
END_METHOD

END_FUNCTION_BLOCK

// ---- 01_PneumaticPress/Io/FB_PressIoCatalog.TcPOU
// Owner-local I/O engineering-data adapter. This is the ONE source for the approved
// tag/address/description/module-role join. It contains no cyclic behavior,
// process-image access, topology algorithms or device logic.
FUNCTION_BLOCK FB_PressIoCatalog
VAR
    _publisher : FB_IoTopologyPublisher;
    _rootPath : STRING(255);
END_VAR

;

METHOD Setup : BOOL
VAR_INPUT
    UnitRef : REFERENCE TO FB_PressDemoUnit;
    // Core §7.5 register. Only its OUTPUT_FORCING gate can mark a channel
    // Forceable, so a production image publishes Forceable=FALSE everywhere and
    // the HMI renders no force affordance at all (§3.9, §10.5.1 rule 1).
    Engineering : REFERENCE TO FB_EngineeringMode;
END_VAR
VAR
    Ok : BOOL;
    SlideIdentity, DoorIdentity, PressIdentity : ST_CylinderIoIdentity;
    PartIdentity, LowAirIdentity, OperatingAirIdentity : ST_IoPointIdentity;
END_VAR
_rootPath := UnitRef.Name;
Ok := _publisher.Setup(DataRef := GVL_PressFieldbus.Topology, ResetData := TRUE);
Ok := _publisher.M_DefineNode(Index := 1, Name := '=000+S-A610-A1',
    DescriptionKey := 'project.hardware.cx2030', TypeId := 'Beckhoff CX2030',
    Address := 'EtherCAT master', ParentIndex := 0) AND Ok;
Ok := _publisher.M_DefineNode(Index := 2, Name := '=000+S-K010',
    DescriptionKey := 'project.hardware.ek1200', TypeId := 'Beckhoff EK1200-5000',
    Address := 'EtherCAT Box 1', ParentIndex := 1) AND Ok;
Ok := _publisher.M_DefineNode(Index := 3, Name := '=000+S-K010B1',
    DescriptionKey := 'project.hardware.el1809', TypeId := 'Beckhoff EL1809',
    Address := 'EtherCAT Box 2', ParentIndex := 2) AND Ok;
Ok := _publisher.M_DefineNode(Index := 4, Name := '=000+S-K010C1',
    DescriptionKey := 'project.hardware.el2809', TypeId := 'Beckhoff EL2809',
    Address := 'EtherCAT Box 3', ParentIndex := 2) AND Ok;
Ok := _publisher.M_DefineNode(Index := 5, Name := '=000+S-K010D1',
    DescriptionKey := 'project.hardware.el6001', TypeId := 'Beckhoff EL6001 RS232',
    Address := 'EtherCAT Box 4', ParentIndex := 2) AND Ok;
Ok := _publisher.M_DefineNode(Index := 6, Name := '=000+S-K010E',
    DescriptionKey := 'project.hardware.el9011', TypeId := 'Beckhoff EL9011',
    Address := 'EtherCAT Box 5', ParentIndex := 2) AND Ok;

// §10.5.1 — the RS232 terminal's process image. It belongs to no module (nothing
// speaks a protocol over it yet), so its ModulePath is the Unit itself: the bus view
// still shows and forces it, and cross-navigation lands somewhere honest.
Ok := _publisher.M_DefineAnalogChannel(NodeIndex := 5, ChannelIndex := 1,
    Tag := '_000K010D1_Status', DescriptionKey := 'project.io.el6001Status',
    Address := '=000+S-K010D1 Status', Path := '=000+S-K010D1/Status',
    ModulePath := _rootPath, Dir := E_ChannelDir.INPUT, EngUnit := '') AND Ok;
Ok := _publisher.M_DefineAnalogChannel(NodeIndex := 5, ChannelIndex := 2,
    Tag := '_000K010D1_DataIn0', DescriptionKey := 'project.io.el6001DataIn',
    Address := '=000+S-K010D1 Data In 0', Path := '=000+S-K010D1/DataIn0',
    ModulePath := _rootPath, Dir := E_ChannelDir.INPUT, EngUnit := '') AND Ok;
Ok := _publisher.M_DefineAnalogChannel(NodeIndex := 5, ChannelIndex := 3,
    Tag := '_000K010D1_DataIn1', DescriptionKey := 'project.io.el6001DataIn',
    Address := '=000+S-K010D1 Data In 1', Path := '=000+S-K010D1/DataIn1',
    ModulePath := _rootPath, Dir := E_ChannelDir.INPUT, EngUnit := '') AND Ok;
Ok := _publisher.M_DefineAnalogChannel(NodeIndex := 5, ChannelIndex := 4,
    Tag := '_000K010D1_DataIn2', DescriptionKey := 'project.io.el6001DataIn',
    Address := '=000+S-K010D1 Data In 2', Path := '=000+S-K010D1/DataIn2',
    ModulePath := _rootPath, Dir := E_ChannelDir.INPUT, EngUnit := '') AND Ok;
Ok := _publisher.M_DefineAnalogChannel(NodeIndex := 5, ChannelIndex := 5,
    Tag := '_000K010D1_Ctrl', DescriptionKey := 'project.io.el6001Ctrl',
    Address := '=000+S-K010D1 Ctrl', Path := '=000+S-K010D1/Ctrl',
    ModulePath := _rootPath, Dir := E_ChannelDir.OUTPUT, EngUnit := '') AND Ok;
Ok := _publisher.M_DefineAnalogChannel(NodeIndex := 5, ChannelIndex := 6,
    Tag := '_000K010D1_DataOut0', DescriptionKey := 'project.io.el6001DataOut',
    Address := '=000+S-K010D1 Data Out 0', Path := '=000+S-K010D1/DataOut0',
    ModulePath := _rootPath, Dir := E_ChannelDir.OUTPUT, EngUnit := '') AND Ok;
Ok := _publisher.M_DefineAnalogChannel(NodeIndex := 5, ChannelIndex := 7,
    Tag := '_000K010D1_DataOut1', DescriptionKey := 'project.io.el6001DataOut',
    Address := '=000+S-K010D1 Data Out 1', Path := '=000+S-K010D1/DataOut1',
    ModulePath := _rootPath, Dir := E_ChannelDir.OUTPUT, EngUnit := '') AND Ok;
Ok := _publisher.M_DefineAnalogChannel(NodeIndex := 5, ChannelIndex := 8,
    Tag := '_000K010D1_DataOut2', DescriptionKey := 'project.io.el6001DataOut',
    Address := '=000+S-K010D1 Data Out 2', Path := '=000+S-K010D1/DataOut2',
    ModulePath := _rootPath, Dir := E_ChannelDir.OUTPUT, EngUnit := '') AND Ok;

Ok := _M_DefineCylinder(Identity := SlideIdentity,
    ModulePath := UnitRef.PartSlide.Name,
    ExtendedSensorTag := '_101B301A', ExtendedSensorDescription := 'project.io.101B301A',
    ExtendedSensorAddress := '=000+S-K010B1 Ch1', ExtendedSensorIndex := 1,
    RetractedSensorTag := '_101B301B', RetractedSensorDescription := 'project.io.101B301B',
    RetractedSensorAddress := '=000+S-K010B1 Ch2', RetractedSensorIndex := 2,
    ExtendOutputTag := '_101K301A', ExtendOutputDescription := 'project.io.101K301A',
    ExtendOutputAddress := '=000+S-K010C1 Ch1', ExtendOutputIndex := 1,
    RetractOutputTag := '_101K301B', RetractOutputDescription := 'project.io.101K301B',
    RetractOutputAddress := '=000+S-K010C1 Ch2', RetractOutputIndex := 2,
    ExtendedTimeoutKey := 'project.error.slideInsideSensorTimeout',
    RetractedTimeoutKey := 'project.error.slideOutsideSensorTimeout',
    BothSensorsKey := 'project.error.slidePositionSensorsConflict') AND Ok;
UnitRef.PartSlide.ConfigureIoIdentity(Identity := SlideIdentity);
Ok := _M_DefineCylinder(Identity := DoorIdentity,
    ModulePath := UnitRef.Door.Name,
    ExtendedSensorTag := '_101B201A', ExtendedSensorDescription := 'project.io.101B201A',
    ExtendedSensorAddress := '=000+S-K010B1 Ch3', ExtendedSensorIndex := 3,
    RetractedSensorTag := '_101B201B', RetractedSensorDescription := 'project.io.101B201B',
    RetractedSensorAddress := '=000+S-K010B1 Ch4', RetractedSensorIndex := 4,
    ExtendOutputTag := '_101K201A', ExtendOutputDescription := 'project.io.101K201A',
    ExtendOutputAddress := '=000+S-K010C1 Ch3', ExtendOutputIndex := 3,
    RetractOutputTag := '_101K201B', RetractOutputDescription := 'project.io.101K201B',
    RetractOutputAddress := '=000+S-K010C1 Ch4', RetractOutputIndex := 4,
    ExtendedTimeoutKey := 'project.error.doorClosedSensorTimeout',
    RetractedTimeoutKey := 'project.error.doorOpenSensorTimeout',
    BothSensorsKey := 'project.error.doorPositionSensorsConflict') AND Ok;
UnitRef.Door.ConfigureIoIdentity(Identity := DoorIdentity);
Ok := _M_DefineCylinder(Identity := PressIdentity,
    ModulePath := UnitRef.PressRam.Name,
    ExtendedSensorTag := '_101B202A', ExtendedSensorDescription := 'project.io.101B202A',
    ExtendedSensorAddress := '=000+S-K010B1 Ch5', ExtendedSensorIndex := 5,
    RetractedSensorTag := '_101B202B', RetractedSensorDescription := 'project.io.101B202B',
    RetractedSensorAddress := '=000+S-K010B1 Ch6', RetractedSensorIndex := 6,
    ExtendOutputTag := '_101K202A', ExtendOutputDescription := 'project.io.101K202A',
    ExtendOutputAddress := '=000+S-K010C1 Ch5', ExtendOutputIndex := 5,
    RetractOutputTag := '_101K202B', RetractOutputDescription := 'project.io.101K202B',
    RetractOutputAddress := '=000+S-K010C1 Ch6', RetractOutputIndex := 6,
    ExtendedTimeoutKey := 'project.error.pressDownSensorTimeout',
    RetractedTimeoutKey := 'project.error.pressUpSensorTimeout',
    BothSensorsKey := 'project.error.pressPositionSensorsConflict') AND Ok;
UnitRef.PressRam.ConfigureIoIdentity(Identity := PressIdentity);

Ok := _M_DefinePoint(NodeIndex := 3, ChannelIndex := 7, Tag := '_101S101',
    DescriptionKey := 'project.io.101S101', Address := '=000+S-K010B1 Ch7',
    ModulePath := UnitRef.TwoHand.Name, Dir := E_ChannelDir.INPUT) AND Ok;
Ok := _M_DefinePoint(NodeIndex := 3, ChannelIndex := 8, Tag := '_101S102',
    DescriptionKey := 'project.io.101S102', Address := '=000+S-K010B1 Ch8',
    ModulePath := UnitRef.TwoHand.Name, Dir := E_ChannelDir.INPUT) AND Ok;
LowAirIdentity.Tag := '_000MB085A_2';
LowAirIdentity.DescriptionKey := 'project.io.000MB085A_2';
LowAirIdentity.Address := '=000+S-K010B1 Ch10';
LowAirIdentity.ModulePath := UnitRef.AirPressureMonitor.Name;
LowAirIdentity.Path := CONCAT(_rootPath, '.IO._000MB085A_2');
Ok := _M_DefineIdentity(NodeIndex := 3, ChannelIndex := 9,
    Identity := LowAirIdentity, Dir := E_ChannelDir.INPUT) AND Ok;
OperatingAirIdentity.Tag := '_000MB085A_4';
OperatingAirIdentity.DescriptionKey := 'project.io.000MB085A_4';
OperatingAirIdentity.Address := '=000+S-K010B1 Ch11';
OperatingAirIdentity.ModulePath := UnitRef.AirPressureMonitor.Name;
OperatingAirIdentity.Path := CONCAT(_rootPath, '.IO._000MB085A_4');
Ok := _M_DefineIdentity(NodeIndex := 3, ChannelIndex := 10,
    Identity := OperatingAirIdentity, Dir := E_ChannelDir.INPUT) AND Ok;
UnitRef.AirPressureMonitor.ConfigureIoIdentity(LowSensor := LowAirIdentity,
    OperatingSensor := OperatingAirIdentity);
PartIdentity.Tag := '_101B601';
PartIdentity.DescriptionKey := 'project.io.101B601';
PartIdentity.Address := '=000+S-K010B1 Ch12';
PartIdentity.ModulePath := UnitRef.PartPresentSensor.Name;
PartIdentity.Path := CONCAT(_rootPath, '.IO._101B601');
Ok := _M_DefineIdentity(NodeIndex := 3, ChannelIndex := 11,
    Identity := PartIdentity, Dir := E_ChannelDir.INPUT) AND Ok;
UnitRef.PartPresentSensor.ConfigureIoIdentity(Identity := PartIdentity);
Ok := _M_DefinePoint(NodeIndex := 3, ChannelIndex := 12, Tag := '_000K911_Y32',
    DescriptionKey := 'project.io.000K911_Y32', Address := '=000+S-K010B1 Ch14',
    ModulePath := UnitRef.PneumaticPower.Name, Dir := E_ChannelDir.INPUT) AND Ok;
Ok := _M_DefinePoint(NodeIndex := 3, ChannelIndex := 13, Tag := '_000K910A',
    DescriptionKey := 'project.io.000K910A', Address := '=000+S-K010B1 Ch15',
    ModulePath := UnitRef.Name, Dir := E_ChannelDir.INPUT) AND Ok;
Ok := _M_DefinePoint(NodeIndex := 4, ChannelIndex := 7, Tag := '_101P101',
    DescriptionKey := 'project.io.101P101', Address := '=000+S-K010C1 Ch7',
    ModulePath := UnitRef.TwoHand.Name, Dir := E_ChannelDir.OUTPUT) AND Ok;
Ok := _M_DefinePoint(NodeIndex := 4, ChannelIndex := 8, Tag := '_101P102',
    DescriptionKey := 'project.io.101P102', Address := '=000+S-K010C1 Ch8',
    ModulePath := UnitRef.TwoHand.Name, Dir := E_ChannelDir.OUTPUT) AND Ok;
Ok := _M_DefinePoint(NodeIndex := 4, ChannelIndex := 9, Tag := '_000K951_A1',
    DescriptionKey := 'project.io.000K951_A1', Address := '=000+S-K010C1 Ch10',
    ModulePath := UnitRef.PneumaticPower.Name, Dir := E_ChannelDir.OUTPUT) AND Ok;
Ok := _M_DefinePoint(NodeIndex := 4, ChannelIndex := 10, Tag := '_000K911_A1',
    DescriptionKey := 'project.io.000K911_A1', Address := '=000+S-K010C1 Ch11',
    ModulePath := UnitRef.PneumaticPower.Name, Dir := E_ChannelDir.OUTPUT) AND Ok;
Ok := _M_DeclareForceable(Engineering := Engineering) AND Ok;
Setup := _publisher.M_Validate() AND Ok;
END_METHOD

// §3.10.2 - the static fieldbus identity this catalog owns (it set the publisher
// up on it), appended to the owning root's manifest. The Unit reaches the
// topology through the catalog it was given, never through the global itself.
METHOD M_AppendTopologyConfig : BOOL
VAR_INPUT
    Pager : REFERENCE TO FB_ConfigPager;
END_VAR
F_AppendTopologyConfig(Topology := GVL_PressFieldbus.Topology, Pager := Pager);
M_AppendTopologyConfig := TRUE;
END_METHOD

// Core §10.5.1 rule 1 — mark the outputs this station allows to be forced from
// the HMI, and ONLY while the §7.5 OUTPUT_FORCING build gate is active.
//
// Two channels of the EL2809 are deliberately excluded even in a commissioning
// image: =000+S-K010C1 Ch10/Ch11 (_000K951_A1 / _000K911_A1) drive the hardwired
// N54 D2 Control On relay chain. That chain is this machine's control-power
// authority, and §10.5.1 rule 4 keeps the standard-PLC force surface out of
// anything with that role. Forcing them would energize control power from a
// diagnostic screen, which is exactly the act this surface must never offer.
METHOD PRIVATE _M_DeclareForceable : BOOL
VAR_INPUT
    Engineering : REFERENCE TO FB_EngineeringMode;
END_VAR
VAR
    c : INT;
    allow : BOOL;
    Ok : BOOL;
END_VAR
Ok := TRUE;
allow := __ISVALIDREF(Engineering) AND_THEN Engineering.ForcingActive;
// Ch1..Ch8: the six valve coils and the two lamps - actuators whose owning CM
// still runs, still holds its interlocks, and reasserts them the moment the Unit
// leaves the idle MANUAL state that made the force effective (§10.5.1 rule 3).
FOR c := 1 TO 8 DO
    Ok := _publisher.M_SetForceable(NodeIndex := 4, ChannelIndex := c,
        Forceable := allow) AND Ok;
END_FOR
_M_DeclareForceable := Ok;
END_METHOD

// Core §10.5.1 — apply one accepted force request to the approved channel join
// this catalog owns (§10.2.1). Every authority check upstream of the physical
// contract has already happened in FB_UnitBase.ForceChannel; the publisher
// rechecks root ownership, OUTPUT direction and the Forceable capability, and
// refuses anything else. This writes only the held set-point: the hardware
// driver decides each scan whether set-points are applied at all.
METHOD M_RouteForce : BOOL
VAR_INPUT
    ChannelPath : STRING(255);
    OwnerRootPath : STRING(255);
    Force : BOOL;
    BoolValue : BOOL;
    AnalogValue : REAL;
END_VAR
M_RouteForce := _publisher.M_SetForce(ChannelPath := ChannelPath,
    OwnerRootPath := OwnerRootPath, Force := Force,
    BoolValue := BoolValue, AnalogValue := AnalogValue);
END_METHOD

METHOD PRIVATE _M_DefineIdentity : BOOL
VAR_INPUT
    NodeIndex : INT;
    ChannelIndex : INT;
    Identity : ST_IoPointIdentity;
    Dir : E_ChannelDir;
END_VAR
_M_DefineIdentity := _publisher.M_DefineDigitalChannel(
    NodeIndex := NodeIndex, ChannelIndex := ChannelIndex, Tag := Identity.Tag,
    DescriptionKey := Identity.DescriptionKey, Address := Identity.Address,
    Path := Identity.Path, ModulePath := Identity.ModulePath, Dir := Dir);
END_METHOD

METHOD PRIVATE _M_DefinePoint : BOOL
VAR_INPUT
    NodeIndex : INT;
    ChannelIndex : INT;
    Tag : STRING(80);
    DescriptionKey : STRING(160);
    Address : STRING(80);
    ModulePath : STRING(255);
    Dir : E_ChannelDir;
END_VAR
VAR
    Path : STRING(255);
END_VAR
Path := CONCAT(_rootPath, CONCAT('.IO.', Tag));
_M_DefinePoint := _publisher.M_DefineDigitalChannel(NodeIndex := NodeIndex,
    ChannelIndex := ChannelIndex, Tag := Tag, DescriptionKey := DescriptionKey,
    Address := Address, Path := Path, ModulePath := ModulePath, Dir := Dir);
END_METHOD

METHOD PRIVATE _M_DefineCylinder : BOOL
VAR_INPUT
    ModulePath : STRING(255);
    ExtendedSensorTag : STRING(80);
    ExtendedSensorDescription : STRING(160);
    ExtendedSensorAddress : STRING(80);
    ExtendedSensorIndex : INT;
    RetractedSensorTag : STRING(80);
    RetractedSensorDescription : STRING(160);
    RetractedSensorAddress : STRING(80);
    RetractedSensorIndex : INT;
    ExtendOutputTag : STRING(80);
    ExtendOutputDescription : STRING(160);
    ExtendOutputAddress : STRING(80);
    ExtendOutputIndex : INT;
    RetractOutputTag : STRING(80);
    RetractOutputDescription : STRING(160);
    RetractOutputAddress : STRING(80);
    RetractOutputIndex : INT;
    ExtendedTimeoutKey : STRING(255);
    RetractedTimeoutKey : STRING(255);
    BothSensorsKey : STRING(255);
END_VAR
VAR_IN_OUT
    Identity : ST_CylinderIoIdentity;
END_VAR
VAR
    Ok : BOOL;
END_VAR
Identity.ExtendedSensor.Tag := ExtendedSensorTag;
Identity.ExtendedSensor.Address := ExtendedSensorAddress;
Identity.ExtendedSensor.DescriptionKey := ExtendedSensorDescription;
Identity.ExtendedSensor.ModulePath := ModulePath;
Identity.ExtendedSensor.Path := CONCAT(_rootPath, CONCAT('.IO.', ExtendedSensorTag));
Identity.RetractedSensor.Tag := RetractedSensorTag;
Identity.RetractedSensor.Address := RetractedSensorAddress;
Identity.RetractedSensor.DescriptionKey := RetractedSensorDescription;
Identity.RetractedSensor.ModulePath := ModulePath;
Identity.RetractedSensor.Path := CONCAT(_rootPath, CONCAT('.IO.', RetractedSensorTag));
Identity.ExtendOutput.Tag := ExtendOutputTag;
Identity.ExtendOutput.Address := ExtendOutputAddress;
Identity.ExtendOutput.DescriptionKey := ExtendOutputDescription;
Identity.ExtendOutput.ModulePath := ModulePath;
Identity.ExtendOutput.Path := CONCAT(_rootPath, CONCAT('.IO.', ExtendOutputTag));
Identity.RetractOutput.Tag := RetractOutputTag;
Identity.RetractOutput.Address := RetractOutputAddress;
Identity.RetractOutput.DescriptionKey := RetractOutputDescription;
Identity.RetractOutput.ModulePath := ModulePath;
Identity.RetractOutput.Path := CONCAT(_rootPath, CONCAT('.IO.', RetractOutputTag));
Identity.ExtendedTimeoutKey := ExtendedTimeoutKey;
Identity.RetractedTimeoutKey := RetractedTimeoutKey;
Identity.BothSensorsKey := BothSensorsKey;
Ok := _publisher.M_DefineDigitalChannel(NodeIndex := 3, ChannelIndex := ExtendedSensorIndex,
    Tag := Identity.ExtendedSensor.Tag, DescriptionKey := Identity.ExtendedSensor.DescriptionKey,
    Address := Identity.ExtendedSensor.Address, Path := Identity.ExtendedSensor.Path,
    ModulePath := ModulePath, Dir := E_ChannelDir.INPUT);
Ok := _publisher.M_DefineDigitalChannel(NodeIndex := 3, ChannelIndex := RetractedSensorIndex,
    Tag := Identity.RetractedSensor.Tag, DescriptionKey := Identity.RetractedSensor.DescriptionKey,
    Address := Identity.RetractedSensor.Address, Path := Identity.RetractedSensor.Path,
    ModulePath := ModulePath, Dir := E_ChannelDir.INPUT) AND Ok;
Ok := _publisher.M_DefineDigitalChannel(NodeIndex := 4, ChannelIndex := ExtendOutputIndex,
    Tag := Identity.ExtendOutput.Tag, DescriptionKey := Identity.ExtendOutput.DescriptionKey,
    Address := Identity.ExtendOutput.Address, Path := Identity.ExtendOutput.Path,
    ModulePath := ModulePath, Dir := E_ChannelDir.OUTPUT) AND Ok;
Ok := _publisher.M_DefineDigitalChannel(NodeIndex := 4, ChannelIndex := RetractOutputIndex,
    Tag := Identity.RetractOutput.Tag, DescriptionKey := Identity.RetractOutput.DescriptionKey,
    Address := Identity.RetractOutput.Address, Path := Identity.RetractOutput.Path,
    ModulePath := ModulePath, Dir := E_ChannelDir.OUTPUT) AND Ok;
_M_DefineCylinder := Ok;
END_METHOD

END_FUNCTION_BLOCK

// ---- 01_PneumaticPress/Sequences/FB_PressDemoHome.TcPOU
// HOME mode chain (Core §6.2/§6.8 ST skeleton on FB_SequenceBase): establish the
// shared load-safe position, then complete. Finite (does not loop).
FUNCTION_BLOCK FB_PressDemoHome EXTENDS FB_SequenceBase
VAR
    {attribute 'OPC.UA.DA' := '0'}
    _outCmd : REFERENCE TO ST_PneumaticPressOutCmd;
    {attribute 'OPC.UA.DA' := '0'}
    _loadPosition : FB_PressDemoLoadPosition;
END_VAR

METHOD M_Run
IF NOT _attached THEN
    RETURN;
END_IF
CASE _step OF
    0:  // initialize
        M_Step(StepNo := 0, StepName := 'project.step.pressHomeInitialize',
            Awaits := 0, AwaitingLabel := '', TimeClass := E_TimeClass.WORK, ExpectedTime := T#0S, Branch := 0);
        _retVal := E_StepResult.ADVANCE;
        M_Advance(OnAdvance := 900, OnJump1 := -1, OnJump2 := -1, OnJump3 := -1);
    900:  // shared load-safe position (composite step, §6.7)
        _retVal := M_RunSub(Chain := _loadPosition, BaseStepNo := 900);
        M_Advance(OnAdvance := 999, OnJump1 := -1, OnJump2 := -1, OnJump3 := -1);
    999:  // complete
        M_Step(StepNo := 999, StepName := 'project.step.pressHomeComplete',
            Awaits := 0, AwaitingLabel := '', TimeClass := E_TimeClass.WORK, ExpectedTime := T#0S, Branch := 0);
        M_Complete();
ELSE
    M_Fault(Reason := E_Reason.STEP_STALLED, DescriptionKey := 'std.error.undefinedStep');
END_CASE
END_METHOD

METHOD Setup : BOOL
VAR_INPUT
    Host : I_SequenceHost;
END_VAR
VAR_IN_OUT
    PressRam : FB_CylinderCM;
    Door : FB_CylinderCM;
    PartSlide : FB_CylinderCM;
    OutCmd : ST_PneumaticPressOutCmd;
END_VAR
_outCmd REF= OutCmd;
Setup := M_Attach(Host := Host) AND __ISVALIDREF(_outCmd)
    AND _loadPosition.Setup(Host := Host, PressRam := PressRam, Door := Door, PartSlide := PartSlide);
END_METHOD

END_FUNCTION_BLOCK

// ---- 01_PneumaticPress/Sequences/FB_PressDemoLoadPosition.TcPOU
// Shared load-safe-position sub-sequence (Core §6.7): ram up, door open, slide
// outside. HOME and CHANGEOVER both embed it as one composite step, passing a
// BaseStepNo window so its detailed progress projects through the Unit's normal
// §6.5 step record. Implemented as a Core §6.8 ST `CASE _step OF` skeleton on
// FB_SequenceBase — the step actions issue child commands only through the §6.1
// handshake (M_TryIssue), and progression rides the shared _retVal via M_Advance.
FUNCTION_BLOCK FB_PressDemoLoadPosition EXTENDS FB_SequenceBase
VAR
    {attribute 'OPC.UA.DA' := '0'}
    _pressRam : REFERENCE TO FB_CylinderCM;
    {attribute 'OPC.UA.DA' := '0'}
    _door : REFERENCE TO FB_CylinderCM;
    {attribute 'OPC.UA.DA' := '0'}
    _partSlide : REFERENCE TO FB_CylinderCM;
END_VAR

// step body runs via M_Run; the Unit calls this instance each scan

